C01837=1110.266,-32.356,-50.134,179.770,5.862,149.113
C01838=1110.271,-32.570,-50.123,179.770,5.858,149.112
C01839=1110.275,-32.820,-50.110,179.770,5.854,149.111
C01840=1110.280,-33.069,-50.097,179.769,5.849,149.110
C01841=1110.285,-33.319,-50.084,179.769,5.845,149.110
C01842=1110.291,-33.570,-50.072,179.769,5.841,149.109
C01843=1110.296,-33.819,-50.059,179.768,5.836,149.108
C01844=1110.301,-34.068,-50.046,179.768,5.832,149.107
C01845=1110.306,-34.318,-50.034,179.768,5.827,149.106
C01846=1110.312,-34.567,-50.021,179.767,5.822,149.105
C01847=1110.316,-34.817,-50.008,179.767,5.818,149.104
C01848=1110.321,-35.067,-49.996,179.766,5.813,149.104
C01849=1110.327,-35.317,-49.983,179.766,5.809,149.103
C01850=1110.332,-35.566,-49.971,179.766,5.805,149.102
C01851=1110.337,-35.816,-49.958,179.765,5.800,149.101
C01852=1110.342,-36.065,-49.945,179.765,5.795,149.100
C01853=1110.348,-36.315,-49.933,179.764,5.790,149.099
C01854=1110.353,-36.564,-49.921,179.763,5.786,149.098
C01855=1110.358,-36.814,-49.908,179.763,5.781,149.097
C01856=1110.362,-37.064,-49.895,179.762,5.777,149.097
C01857=1110.368,-37.314,-49.883,179.762,5.772,149.096
C01858=1110.374,-37.563,-49.870,179.762,5.767,149.095
C01859=1110.379,-37.813,-49.857,179.761,5.762,149.094
C01860=1110.384,-38.062,-49.845,179.760,5.758,149.093
C01861=1110.389,-38.312,-49.833,179.760,5.753,149.092
C01862=1110.394,-38.562,-49.820,179.759,5.749,149.091
C01863=1110.399,-38.811,-49.807,179.759,5.744,149.090
C01864=1110.404,-39.061,-49.795,179.758,5.739,149.089
C01865=1110.409,-39.311,-49.783,179.758,5.734,149.089
C01866=1110.415,-39.560,-49.770,179.758,5.730,149.088
C01867=1110.420,-39.810,-49.758,179.757,5.725,149.087
C01868=1110.425,-40.059,-49.746,179.756,5.719,149.086
C01869=1110.430,-40.309,-49.733,179.756,5.715,149.085
C01870=1110.435,-40.559,-49.721,179.755,5.710,149.084
C01871=1110.440,-40.808,-49.708,179.754,5.705,149.083
C01872=1110.446,-41.058,-49.696,179.753,5.700,149.082
C01873=1110.451,-41.308,-49.684,179.753,5.695,149.082
C01874=1110.456,-41.557,-49.671,179.752,5.690,149.081
C01875=1110.461,-41.807,-49.659,179.752,5.684,149.079
C01876=1110.466,-42.056,-49.647,179.751,5.680,149.079
C01877=1110.472,-42.306,-49.635,179.751,5.675,149.078
C01878=1110.476,-42.556,-49.622,179.750,5.669,149.077
C01879=1110.482,-42.806,-49.610,179.749,5.665,149.076
C01880=1110.486,-43.055,-49.598,179.749,5.660,149.075
C01881=1110.492,-43.305,-49.586,179.749,5.655,149.074
C01882=1110.497,-43.554,-49.573,179.750,5.651,149.073
C01883=1110.502,-43.804,-49.561,179.750,5.645,149.071
C01884=1110.507,-44.054,-49.549,179.750,5.640,149.070
C01885=1110.513,-44.304,-49.537,179.750,5.636,149.069
C01886=1110.518,-44.553,-49.524,179.750,5.631,149.068
C01887=1110.522,-44.768,-49.514,179.750,5.627,149.067
C01888=1110.526,-44.982,-49.504,179.750,5.623,149.066
C01889=1110.531,-45.197,-49.493,179.751,5.619,149.066
C01890=1110.535,-45.411,-49.482,179.751,5.615,149.065
C01891=1110.540,-45.626,-49.472,179.751,5.612,149.064
C01892=1110.545,-45.840,-49.463,179.751,5.608,149.063
C01893=1110.549,-46.055,-49.452,179.751,5.603,149.062
C01894=1110.554,-46.270,-49.441,179.751,5.598,149.061
C01895=1110.559,-46.519,-49.429,179.751,5.595,149.060
C01896=1110.564,-46.769,-49.418,179.752,5.589,149.059
C01897=1110.569,-47.019,-49.406,179.752,5.584,149.058
C01898=1110.574,-47.268,-49.393,179.752,5.580,149.057
C01899=1110.580,-47.518,-49.381,179.752,5.575,149.055
C01900=1110.585,-47.767,-49.369,179.753,5.571,149.054
C01901=1110.589,-48.017,-49.357,179.753,5.566,149.053
C01902=1110.595,-48.267,-49.345,179.752,5.561,149.052
C01903=1110.600,-48.516,-49.333,179.753,5.557,149.051
C01904=1110.605,-48.766,-49.321,179.753,5.552,149.050
C01905=1110.611,-49.016,-49.309,179.753,5.548,149.049
C01906=1110.615,-49.265,-49.297,179.753,5.542,149.048
C01907=1110.621,-49.515,-49.285,179.753,5.537,149.047
C01908=1110.626,-49.765,-49.273,179.753,5.533,149.046
C01909=1110.631,-50.014,-49.261,179.753,5.528,149.045
C01910=1110.636,-50.264,-49.249,179.754,5.523,149.043
C01911=1110.641,-50.514,-49.237,179.754,5.519,149.042
C01912=1110.647,-50.764,-49.226,179.754,5.514,149.041
C01913=1110.652,-51.013,-49.213,179.754,5.509,149.040
C01914=1110.656,-51.263,-49.202,179.755,5.505,149.039
C01915=1110.662,-51.513,-49.190,179.754,5.500,149.038
C01916=1110.667,-51.763,-49.178,179.755,5.496,149.037
C01917=1110.672,-52.012,-49.165,179.755,5.490,149.036
C01918=1110.677,-52.261,-49.154,179.755,5.486,149.035
C01919=1110.683,-52.511,-49.142,179.755,5.481,149.034
C01920=1110.688,-52.761,-49.130,179.755,5.476,149.033
C01921=1110.692,-53.010,-49.118,179.755,5.471,149.032
C01922=1110.698,-53.260,-49.106,179.756,5.467,149.031
C01923=1110.704,-53.510,-49.095,179.756,5.462,149.029
C01924=1110.709,-53.759,-49.083,179.756,5.458,149.029
C01925=1110.714,-54.009,-49.072,179.756,5.453,149.027
C01926=1110.719,-54.258,-49.059,179.756,5.448,149.026
C01927=1110.725,-54.508,-49.047,179.756,5.444,149.025
C01928=1110.729,-54.758,-49.036,179.756,5.439,149.024
C01929=1110.735,-55.008,-49.024,179.756,5.434,149.023
C01930=1110.740,-55.258,-49.012,179.757,5.430,149.022
C01931=1110.745,-55.507,-49.001,179.757,5.425,149.021
C01932=1110.750,-55.757,-48.989,179.757,5.421,149.020
C01933=1110.755,-56.006,-48.977,179.757,5.415,149.019
C01934=1110.761,-56.256,-48.965,179.757,5.410,149.018
C01935=1110.766,-56.506,-48.954,179.757,5.406,149.017
C01936=1110.771,-56.755,-48.942,179.757,5.401,149.016
C01937=1110.776,-57.005,-48.930,179.757,5.396,149.014
C01938=1110.781,-57.255,-48.919,179.758,5.392,149.014
C01939=1110.786,-57.505,-48.907,179.758,5.387,149.012
C01940=1110.792,-57.755,-48.895,179.757,5.382,149.011
C01941=1110.796,-58.004,-48.884,179.758,5.378,149.010
C01942=1110.802,-58.253,-48.872,179.758,5.373,149.009
C01943=1110.807,-58.468,-48.862,179.758,5.369,149.008
C01944=1110.811,-58.683,-48.852,179.758,5.365,149.007
C01945=1110.815,-58.898,-48.842,179.758,5.361,149.007
C01946=1110.820,-59.112,-48.832,179.758,5.357,149.006
C01947=1110.824,-59.326,-48.822,179.759,5.353,149.005
C01948=1110.829,-59.541,-48.812,179.758,5.349,149.004
C01949=1110.833,-59.756,-48.802,179.758,5.345,149.003
C01950=1110.837,-59.971,-48.792,179.759,5.341,149.002
C01951=1110.843,-60.220,-48.781,179.758,5.336,149.001
C01952=1110.848,-60.470,-48.769,179.758,5.331,149.000
C01953=1110.853,-60.720,-48.758,179.758,5.326,148.999
C01954=1110.858,-60.969,-48.746,179.757,5.321,148.998
C01955=1110.863,-61.219,-48.735,179.757,5.316,148.997
C01956=1110.869,-61.470,-48.724,179.757,5.311,148.996
C01957=1110.874,-61.719,-48.713,179.756,5.306,148.995
C01958=1110.879,-61.969,-48.701,179.755,5.300,148.994
C01959=1110.884,-62.218,-48.690,179.755,5.296,148.993
C01960=1110.890,-62.468,-48.678,179.755,5.291,148.992
C01961=1110.895,-62.717,-48.667,179.755,5.286,148.991
C01962=1110.900,-62.967,-48.655,179.754,5.281,148.990
C01963=1110.905,-63.217,-48.644,179.754,5.275,148.989
C01964=1110.910,-63.466,-48.632,179.753,5.270,148.988
C01965=1110.915,-63.716,-48.620,179.753,5.265,148.987
C01966=1110.921,-63.966,-48.610,179.753,5.260,148.986
C01967=1110.926,-64.216,-48.598,179.753,5.256,148.985
C01968=1110.931,-64.465,-48.587,179.752,5.250,148.984
C01969=1110.936,-64.715,-48.575,179.752,5.245,148.983
C01970=1110.942,-64.964,-48.564,179.752,5.240,148.982
C01971=1110.947,-65.214,-48.554,179.752,5.235,148.981
C01972=1110.952,-65.464,-48.542,179.752,5.230,148.980
C01973=1110.957,-65.713,-48.531,179.751,5.224,148.979
C01974=1110.963,-65.963,-48.519,179.751,5.219,148.978
C01975=1110.967,-66.213,-48.508,179.750,5.214,148.977
C01976=1110.972,-66.463,-48.497,179.751,5.209,148.976
C01977=1110.978,-66.712,-48.486,179.751,5.204,148.974
C01978=1110.983,-66.962,-48.474,179.750,5.199,148.973
C01979=1110.988,-67.212,-48.464,179.750,5.194,148.972
C01980=1110.994,-67.461,-48.452,179.750,5.189,148.971
C01981=1110.999,-67.711,-48.441,179.750,5.184,148.970
C01982=1111.004,-67.961,-48.430,179.750,5.178,148.969
C01983=1111.010,-68.210,-48.419,179.749,5.174,148.968
C01984=1111.015,-68.460,-48.407,179.749,5.168,148.967
C01985=1111.019,-68.710,-48.396,179.749,5.163,148.966
C01986=1111.026,-68.960,-48.385,179.749,5.158,148.965
C01987=1111.030,-69.209,-48.374,179.749,5.153,148.964
C01988=1111.035,-69.459,-48.364,179.749,5.148,148.963
C01989=1111.041,-69.709,-48.352,179.749,5.143,148.962
C01990=1111.046,-69.958,-48.341,179.749,5.138,148.960
C01991=1111.051,-70.209,-48.330,179.748,5.132,148.959
C01992=1111.056,-70.457,-48.319,179.748,5.127,148.958
C01993=1111.062,-70.707,-48.307,179.748,5.122,148.957
C01994=1111.067,-70.958,-48.297,179.748,5.117,148.956
C01995=1111.072,-71.207,-48.286,179.748,5.112,148.955
C01996=1111.077,-71.457,-48.275,179.748,5.106,148.954
C01997=1111.083,-71.706,-48.264,179.749,5.101,148.953
C01998=1111.088,-71.956,-48.253,179.748,5.097,148.952
C01999=1111.092,-72.171,-48.243,179.748,5.091,148.950
C02000=1111.097,-72.385,-48.234,179.748,5.087,148.950
C02001=1111.101,-72.601,-48.225,179.748,5.083,148.949
C02002=1111.106,-72.815,-48.215,179.748,5.078,148.948
C02003=1111.110,-73.030,-48.206,179.748,5.074,148.947
C02004=1111.114,-73.245,-48.196,179.748,5.069,148.946
C02005=1111.120,-73.459,-48.188,179.748,5.065,148.945
C02006=1111.124,-73.674,-48.178,179.748,5.060,148.944
C02007=1111.130,-73.924,-48.167,179.748,5.055,148.943
C02008=1111.134,-74.174,-48.156,179.748,5.050,148.941
C02009=1111.140,-74.423,-48.146,179.748,5.045,148.940
C02010=1111.145,-74.673,-48.135,179.748,5.040,148.939
C02011=1111.150,-74.923,-48.124,179.748,5.035,148.938
C02012=1111.156,-75.172,-48.112,179.748,5.030,148.937
C02013=1111.161,-75.422,-48.102,179.749,5.024,148.936
C02014=1111.166,-75.671,-48.091,179.749,5.019,148.935
C02015=1111.171,-75.922,-48.080,179.749,5.014,148.933
C02016=1111.176,-76.171,-48.070,179.749,5.009,148.932
C02017=1111.181,-76.421,-48.059,179.749,5.004,148.931
C02018=1111.187,-76.670,-48.049,179.749,4.999,148.930
C02019=1111.192,-76.921,-48.038,179.749,4.994,148.929
C02020=1111.198,-77.170,-48.027,179.750,4.988,148.928
C02021=1111.203,-77.420,-48.016,179.750,4.983,148.926
C02022=1111.208,-77.669,-48.005,179.750,4.978,148.925
C02023=1111.213,-77.919,-47.995,179.750,4.973,148.924
C02024=1111.219,-78.169,-47.984,179.750,4.968,148.923
C02025=1111.224,-78.419,-47.974,179.750,4.963,148.922
C02026=1111.229,-78.668,-47.963,179.751,4.958,148.920
C02027=1111.234,-78.918,-47.952,179.751,4.952,148.919
C02028=1111.240,-79.168,-47.942,179.751,4.947,148.918
C02029=1111.244,-79.417,-47.931,179.751,4.942,148.917
C02030=1111.250,-79.667,-47.921,179.751,4.937,148.916
C02031=1111.256,-79.917,-47.909,179.751,4.932,148.915
C02032=1111.261,-80.167,-47.899,179.752,4.927,148.913
C02033=1111.266,-80.417,-47.888,179.752,4.922,148.912
C02034=1111.271,-80.666,-47.878,179.752,4.916,148.911
C02035=1111.276,-80.916,-47.867,179.752,4.911,148.910
C02036=1111.282,-81.166,-47.857,179.752,4.906,148.909
C02037=1111.287,-81.415,-47.846,179.753,4.901,148.907
C02038=1111.292,-81.665,-47.835,179.753,4.895,148.906
C02039=1111.298,-81.915,-47.825,179.753,4.890,148.905
C02040=1111.303,-82.165,-47.815,179.753,4.885,148.904
C02041=1111.308,-82.414,-47.804,179.754,4.880,148.903
C02042=1111.313,-82.664,-47.794,179.754,4.876,148.901
C02043=1111.318,-82.913,-47.783,179.754,4.871,148.900
C02044=1111.323,-83.164,-47.773,179.755,4.865,148.899
C02045=1111.329,-83.413,-47.763,179.755,4.860,148.898
C02046=1111.334,-83.663,-47.752,179.755,4.855,148.897
C02047=1111.339,-83.913,-47.742,179.756,4.850,148.895
C02048=1111.345,-84.162,-47.731,179.756,4.844,148.894
C02049=1111.350,-84.412,-47.720,179.756,4.839,148.893
C02050=1111.355,-84.662,-47.710,179.757,4.835,148.892
C02051=1111.361,-84.911,-47.700,179.757,4.830,148.891
C02052=1111.366,-85.161,-47.689,179.757,4.825,148.889
C02053=1111.371,-85.411,-47.679,179.757,4.819,148.888
C02054=1111.376,-85.661,-47.669,179.757,4.814,148.887
C02055=1111.381,-85.876,-47.660,179.758,4.810,148.886
C02056=1111.385,-86.090,-47.650,179.758,4.806,148.885
C02057=1111.390,-86.305,-47.642,179.759,4.801,148.884
C02058=1111.395,-86.520,-47.633,179.759,4.797,148.883
C02059=1111.399,-86.735,-47.624,179.759,4.793,148.882
C02060=1111.403,-86.949,-47.616,179.760,4.789,148.881
C02061=1111.408,-87.165,-47.607,179.760,4.784,148.880
C02062=1111.412,-87.379,-47.598,179.760,4.780,148.879
C02063=1111.417,-87.629,-47.587,179.761,4.774,148.877
C02064=1111.423,-87.878,-47.577,179.761,4.770,148.876
C02065=1111.428,-88.128,-47.567,179.762,4.765,148.875
C02066=1111.433,-88.378,-47.556,179.762,4.760,148.874
C02067=1111.438,-88.627,-47.547,179.763,4.755,148.873
C02068=1111.444,-88.877,-47.536,179.763,4.750,148.871
C02069=1111.449,-89.127,-47.526,179.763,4.745,148.870
C02070=1111.454,-89.377,-47.516,179.764,4.740,148.869
C02071=1111.460,-89.626,-47.505,179.764,4.735,148.868
C02072=1111.465,-89.877,-47.495,179.765,4.730,148.866
C02073=1111.470,-90.126,-47.485,179.765,4.725,148.865
C02074=1111.476,-90.376,-47.476,179.766,4.721,148.864
C02075=1111.481,-90.626,-47.465,179.766,4.715,148.863
C02076=1111.486,-90.876,-47.455,179.766,4.710,148.861
C02077=1111.492,-91.125,-47.445,179.767,4.706,148.860
C02078=1111.496,-91.375,-47.435,179.767,4.700,148.859
C02079=1111.502,-91.625,-47.424,179.768,4.695,148.858
C02080=1111.507,-91.874,-47.414,179.768,4.691,148.857
C02081=1111.512,-92.125,-47.404,179.769,4.686,148.856
C02082=1111.517,-92.374,-47.394,179.769,4.681,148.854
C02083=1111.523,-92.623,-47.384,179.770,4.676,148.853
C02084=1111.529,-92.873,-47.374,179.770,4.671,148.852
C02085=1111.534,-93.124,-47.364,179.771,4.666,148.851
C02086=1111.539,-93.373,-47.354,179.771,4.661,148.849
C02087=1111.544,-93.623,-47.344,179.772,4.657,148.848
C02088=1111.549,-93.873,-47.333,179.772,4.652,148.847
C02089=1111.555,-94.122,-47.323,179.773,4.647,148.846
C02090=1111.560,-94.372,-47.314,179.773,4.642,148.845
C02091=1111.565,-94.621,-47.303,179.773,4.637,148.843
C02092=1111.571,-94.872,-47.293,179.774,4.633,148.842
C02093=1111.576,-95.121,-47.284,179.774,4.628,148.841
C02094=1111.581,-95.371,-47.274,179.775,4.622,148.840
C02095=1111.587,-95.620,-47.263,179.775,4.617,148.839
C02096=1111.592,-95.871,-47.253,179.776,4.613,148.837
C02097=1111.597,-96.120,-47.244,179.776,4.608,148.836
C02098=1111.602,-96.370,-47.234,179.776,4.603,148.835
C02099=1111.608,-96.619,-47.224,179.777,4.598,148.834
C02100=1111.613,-96.869,-47.214,179.777,4.593,148.833
C02101=1111.618,-97.120,-47.204,179.777,4.588,148.832
C02102=1111.624,-97.369,-47.194,179.777,4.583,148.830
C02103=1111.629,-97.618,-47.184,179.778,4.578,148.829
C02104=1111.634,-97.868,-47.174,179.779,4.573,148.828
C02105=1111.640,-98.119,-47.164,179.779,4.568,148.827
C02106=1111.644,-98.368,-47.155,179.779,4.563,148.826
C02107=1111.650,-98.618,-47.144,179.780,4.559,148.824
C02108=1111.655,-98.867,-47.135,179.780,4.553,148.823
C02109=1111.661,-99.117,-47.125,179.780,4.548,148.822
C02110=1111.666,-99.367,-47.115,179.780,4.543,148.821
C02111=1111.670,-99.582,-47.106,179.781,4.539,148.820
C02112=1111.675,-99.796,-47.098,179.781,4.535,148.819
C02113=1111.679,-100.012,-47.090,179.781,4.531,148.818
C02114=1111.684,-100.227,-47.081,179.782,4.527,148.817
C02115=1111.689,-100.441,-47.073,179.782,4.522,148.816
C02116=1111.693,-100.656,-47.064,179.782,4.518,148.815
C02117=1111.698,-100.871,-47.056,179.783,4.514,148.814
C02118=1111.703,-101.086,-47.048,179.783,4.510,148.813
C02119=1111.708,-101.335,-47.038,179.783,4.505,148.811
C02120=1111.714,-101.586,-47.028,179.784,4.500,148.810
C02121=1111.718,-101.836,-47.018,179.784,4.494,148.809
C02122=1111.723,-102.085,-47.008,179.785,4.490,148.808
C02123=1111.729,-102.335,-46.999,179.785,4.485,148.807
C02124=1111.734,-102.584,-46.989,179.785,4.480,148.805
C02125=1111.739,-102.834,-46.980,179.785,4.475,148.804
C02126=1111.745,-103.084,-46.970,179.786,4.469,148.803
C02127=1111.751,-103.333,-46.960,179.786,4.465,148.802
C02128=1111.755,-103.584,-46.951,179.787,4.460,148.801
C02129=1111.761,-103.834,-46.940,179.787,4.455,148.799
C02130=1111.766,-104.083,-46.931,179.787,4.450,148.798
C02131=1111.771,-104.333,-46.921,179.787,4.444,148.797
C02132=1111.777,-104.583,-46.912,179.788,4.440,148.796
C02133=1111.782,-104.832,-46.902,179.788,4.435,148.795
C02134=1111.787,-105.082,-46.893,179.789,4.430,148.794
C02135=1111.792,-105.331,-46.884,179.789,4.425,148.792
C02136=1111.798,-105.582,-46.874,179.789,4.420,148.791
C02137=1111.802,-105.831,-46.864,179.790,4.415,148.790
C02138=1111.808,-106.082,-46.855,179.790,4.410,148.789
C02139=1111.813,-106.331,-46.845,179.790,4.405,148.788
C02140=1111.819,-106.581,-46.836,179.791,4.400,148.786
C02141=1111.824,-106.830,-46.826,179.791,4.395,148.785
C02142=1111.830,-107.080,-46.816,179.791,4.389,148.784
C02143=1111.835,-107.330,-46.807,179.792,4.385,148.783
C02144=1111.841,-107.580,-46.797,179.792,4.380,148.782
C02145=1111.845,-107.829,-46.788,179.792,4.375,148.780
C02146=1111.851,-108.079,-46.779,179.793,4.370,148.779
C02147=1111.857,-108.329,-46.769,179.793,4.364,148.778
C02148=1111.861,-108.579,-46.759,179.793,4.359,148.777
C02149=1111.867,-108.829,-46.750,179.794,4.355,148.775
C02150=1111.872,-109.078,-46.740,179.795,4.349,148.774
C02151=1111.877,-109.328,-46.731,179.795,4.344,148.773
C02152=1111.883,-109.578,-46.722,179.795,4.339,148.772
C02153=1111.888,-109.828,-46.712,179.795,4.334,148.770
C02154=1111.893,-110.078,-46.703,179.796,4.329,148.769
C02155=1111.898,-110.327,-46.693,179.796,4.324,148.768
C02156=1111.903,-110.577,-46.684,179.796,4.318,148.767
C02157=1111.909,-110.827,-46.675,179.797,4.314,148.766
C02158=1111.914,-111.076,-46.665,179.797,4.309,148.764
C02159=1111.919,-111.326,-46.656,179.798,4.304,148.763
C02160=1111.925,-111.576,-46.647,179.798,4.299,148.762
C02161=1111.930,-111.826,-46.637,179.798,4.293,148.761
C02162=1111.935,-112.075,-46.628,179.799,4.288,148.759
C02163=1111.941,-112.326,-46.619,179.799,4.283,148.758
C02164=1111.946,-112.575,-46.610,179.799,4.278,148.757
C02165=1111.951,-112.825,-46.600,179.800,4.272,148.756
C02166=1111.957,-113.075,-46.591,179.800,4.267,148.755
C02167=1111.962,-113.290,-46.583,179.800,4.263,148.754
C02168=1111.966,-113.504,-46.575,179.801,4.259,148.752
C02169=1111.971,-113.719,-46.567,179.801,4.254,148.751
C02170=1111.975,-113.935,-46.559,179.802,4.250,148.750
C02171=1111.980,-114.150,-46.551,179.802,4.246,148.749
C02172=1111.985,-114.365,-46.543,179.802,4.241,148.748
C02173=1111.989,-114.579,-46.535,179.803,4.237,148.747
C02174=1111.994,-114.794,-46.527,179.802,4.232,148.746
C02175=1111.999,-115.044,-46.518,179.803,4.228,148.745
C02176=1112.004,-115.294,-46.510,179.804,4.222,148.743
C02177=1112.010,-115.544,-46.499,179.804,4.217,148.742
C02178=1112.015,-115.793,-46.490,179.804,4.212,148.741
C02179=1112.020,-116.043,-46.482,179.805,4.207,148.740
C02180=1112.026,-116.293,-46.473,179.805,4.201,148.739
C02181=1112.031,-116.543,-46.463,179.805,4.196,148.737
C02182=1112.037,-116.793,-46.454,179.806,4.191,148.736
C02183=1112.041,-117.042,-46.445,179.806,4.185,148.735
C02184=1112.047,-117.292,-46.436,179.807,4.180,148.733
C02185=1112.052,-117.542,-46.427,179.807,4.175,148.732
C02186=1112.058,-117.792,-46.417,179.807,4.170,148.731
C02187=1112.063,-118.041,-46.409,179.808,4.164,148.730
C02188=1112.069,-118.291,-46.400,179.808,4.159,148.728
C02189=1112.074,-118.541,-46.391,179.809,4.154,148.727
C02190=1112.079,-118.791,-46.382,179.809,4.149,148.726
C02191=1112.085,-119.041,-46.373,179.809,4.144,148.725
C02192=1112.090,-119.290,-46.363,179.810,4.138,148.723
C02193=1112.095,-119.540,-46.354,179.810,4.133,148.722
C02194=1112.100,-119.790,-46.345,179.810,4.128,148.721
C02195=1112.105,-120.040,-46.336,179.811,4.123,148.720
C02196=1112.111,-120.289,-46.328,179.812,4.117,148.718
C02197=1112.117,-120.539,-46.318,179.812,4.112,148.717
C02198=1112.122,-120.789,-46.309,179.812,4.107,148.716
C02199=1112.127,-121.039,-46.301,179.812,4.102,148.715
C02200=1112.132,-121.289,-46.292,179.813,4.096,148.713
C02201=1112.138,-121.539,-46.283,179.813,4.091,148.712
C02202=1112.143,-121.789,-46.274,179.814,4.086,148.711
C02203=1112.149,-122.038,-46.265,179.814,4.081,148.709
C02204=1112.154,-122.288,-46.256,179.814,4.074,148.708
C02205=1112.159,-122.537,-46.247,179.815,4.069,148.707
C02206=1112.165,-122.788,-46.238,179.815,4.064,148.706
C02207=1112.174,-123.205,-46.223,179.816,4.056,148.703
C02208=1112.182,-123.622,-46.209,179.817,4.047,148.701
C02209=1112.191,-124.039,-46.194,179.817,4.037,148.699
C02210=1112.200,-124.456,-46.179,179.818,4.028,148.697
C02211=1112.205,-124.706,-46.170,179.818,4.023,148.696
C02212=1112.211,-124.957,-46.162,179.819,4.018,148.694
C02213=1112.216,-125.206,-46.153,179.819,4.012,148.693
C02214=1112.222,-125.456,-46.145,179.820,4.007,148.692
C02215=1112.227,-125.705,-46.136,179.820,4.001,148.690
C02216=1112.232,-125.955,-46.127,179.820,3.996,148.689
C02217=1112.237,-126.205,-46.118,179.821,3.991,148.688
C02218=1112.242,-126.455,-46.109,179.821,3.985,148.686
C02219=1112.248,-126.704,-46.101,179.822,3.980,148.685
C02220=1112.254,-126.955,-46.092,179.822,3.974,148.684
C02221=1112.259,-127.204,-46.084,179.823,3.969,148.682
C02222=1112.264,-127.454,-46.075,179.823,3.963,148.681
C02223=1112.270,-127.717,-46.065,179.823,3.958,148.680
C02224=1112.276,-127.979,-46.057,179.824,3.952,148.678
C02225=1112.282,-128.242,-46.047,179.824,3.946,148.677
C02226=1112.287,-128.504,-46.038,179.825,3.940,148.676
C02227=1111.864,-128.495,-46.065,179.832,3.945,148.674
C02228=1111.859,-128.280,-46.072,179.832,3.949,148.675
C02229=1111.855,-128.065,-46.079,179.831,3.954,148.677
C02230=1111.850,-127.850,-46.086,179.831,3.958,148.677
C02231=1111.845,-127.634,-46.094,179.831,3.963,148.679
C02232=1111.841,-127.419,-46.102,179.830,3.968,148.680
C02233=1111.837,-127.205,-46.109,179.830,3.973,148.681
C02234=1111.832,-126.990,-46.117,179.830,3.978,148.682
C02235=1111.827,-126.775,-46.124,179.829,3.982,148.683
C02236=1111.822,-126.525,-46.133,179.828,3.987,148.685
C02237=1111.817,-126.275,-46.142,179.828,3.993,148.686
C02238=1111.811,-126.026,-46.150,179.828,3.999,148.687
C02239=1111.806,-125.776,-46.159,179.828,4.004,148.688
C02240=1111.800,-125.526,-46.168,179.827,4.009,148.690
C02241=1111.795,-125.276,-46.177,179.826,4.015,148.691
C02242=1111.790,-125.026,-46.186,179.826,4.020,148.692
C02243=1111.784,-124.777,-46.194,179.825,4.025,148.694
C02244=1111.779,-124.527,-46.203,179.825,4.031,148.695
C02245=1111.774,-124.277,-46.212,179.824,4.036,148.697
C02246=1111.769,-124.027,-46.220,179.824,4.041,148.698
C02247=1111.763,-123.777,-46.230,179.824,4.047,148.699
C02248=1111.757,-123.528,-46.238,179.823,4.053,148.700
C02249=1111.752,-123.278,-46.247,179.823,4.058,148.702
C02250=1111.747,-123.028,-46.256,179.823,4.063,148.703
C02251=1111.741,-122.778,-46.265,179.823,4.068,148.704
C02252=1111.736,-122.528,-46.274,179.822,4.074,148.706
C02253=1111.731,-122.278,-46.283,179.821,4.079,148.707
C02254=1111.726,-122.028,-46.292,179.821,4.084,148.708
C02255=1111.720,-121.779,-46.300,179.820,4.090,148.709
C02256=1111.715,-121.529,-46.309,179.820,4.095,148.711
C02257=1111.709,-121.279,-46.319,179.820,4.100,148.712
C02258=1111.704,-121.029,-46.327,179.820,4.105,148.713
C02259=1111.699,-120.780,-46.336,179.819,4.111,148.715
C02260=1111.694,-120.530,-46.346,179.818,4.116,148.716
C02261=1111.689,-120.280,-46.355,179.818,4.121,148.717
C02262=1111.683,-120.031,-46.364,179.817,4.127,148.718
C02263=1111.677,-119.781,-46.373,179.817,4.132,148.720
C02264=1111.672,-119.531,-46.382,179.817,4.137,148.721
C02265=1111.667,-119.281,-46.391,179.816,4.142,148.722
C02266=1111.661,-119.032,-46.400,179.816,4.147,148.723
C02267=1111.656,-118.782,-46.408,179.815,4.153,148.725
C02268=1111.650,-118.532,-46.418,179.815,4.158,148.726
C02269=1111.645,-118.282,-46.427,179.815,4.163,148.727
C02270=1111.640,-118.033,-46.436,179.815,4.168,148.728
C02271=1111.635,-117.783,-46.445,179.814,4.174,148.730
C02272=1111.630,-117.533,-46.454,179.814,4.179,148.731
C02273=1111.624,-117.283,-46.464,179.813,4.184,148.732
C02274=1111.619,-117.033,-46.473,179.813,4.189,148.733
C02275=1111.613,-116.784,-46.481,179.813,4.194,148.735
C02276=1111.608,-116.534,-46.491,179.812,4.200,148.736
C02277=1111.602,-116.284,-46.500,179.812,4.205,148.737
C02278=1111.597,-116.034,-46.509,179.811,4.210,148.739
C02279=1111.592,-115.785,-46.518,179.811,4.215,148.740
C02280=1111.587,-115.535,-46.527,179.811,4.221,148.741
C02281=1111.581,-115.285,-46.537,179.811,4.226,148.742
C02282=1111.576,-115.035,-46.546,179.810,4.231,148.743
C02283=1111.571,-114.785,-46.555,179.810,4.237,148.745
C02284=1111.566,-114.570,-46.563,179.809,4.240,148.746
C02285=1111.562,-114.356,-46.571,179.809,4.244,148.747
C02286=1111.557,-114.140,-46.579,179.809,4.250,148.748
C02287=1111.553,-113.926,-46.587,179.808,4.254,148.749
C02288=1111.548,-113.711,-46.595,179.808,4.259,148.750
C02289=1111.543,-113.495,-46.602,179.808,4.263,148.751
C02290=1111.539,-113.281,-46.611,179.807,4.267,148.752
C02291=1111.535,-113.065,-46.619,179.807,4.272,148.753
C02292=1111.529,-112.816,-46.629,179.807,4.277,148.754
C02293=1111.524,-112.566,-46.638,179.807,4.282,148.756
C02294=1111.519,-112.316,-46.647,179.806,4.287,148.757
C02295=1111.513,-112.066,-46.657,179.805,4.292,148.758
C02296=1111.508,-111.817,-46.666,179.805,4.297,148.760
C02297=1111.503,-111.567,-46.675,179.804,4.302,148.761
C02298=1111.497,-111.317,-46.685,179.804,4.308,148.762
C02299=1111.492,-111.067,-46.694,179.804,4.313,148.763
C02300=1111.486,-110.817,-46.703,179.804,4.318,148.764
C02301=1111.481,-110.568,-46.713,179.803,4.323,148.766
C02302=1111.476,-110.318,-46.722,179.803,4.327,148.767
C02303=1111.470,-110.068,-46.731,179.802,4.333,148.768
C02304=1111.465,-109.819,-46.741,179.802,4.338,148.769
C02305=1111.459,-109.568,-46.750,179.802,4.343,148.770
C02306=1111.455,-109.319,-46.760,179.802,4.348,148.772
C02307=1111.449,-109.069,-46.769,179.801,4.353,148.773
C02308=1111.443,-108.819,-46.778,179.801,4.359,148.774
C02309=1111.439,-108.570,-46.788,179.800,4.364,148.775
C02310=1111.433,-108.320,-46.798,179.800,4.368,148.777
C02311=1111.428,-108.071,-46.807,179.799,4.373,148.778
C02312=1111.423,-107.821,-46.816,179.799,4.379,148.779
C02313=1111.417,-107.571,-46.826,179.799,4.384,148.780
C02314=1111.413,-107.321,-46.836,179.799,4.389,148.781
C02315=1111.407,-107.071,-46.846,179.798,4.394,148.783
C02316=1111.402,-106.821,-46.855,179.797,4.398,148.784
C02317=1111.396,-106.572,-46.865,179.797,4.403,148.785
C02318=1111.391,-106.322,-46.874,179.797,4.409,148.786
C02319=1111.385,-106.072,-46.884,179.797,4.414,148.787
C02320=1111.380,-105.822,-46.893,179.797,4.419,148.789
C02321=1111.375,-105.573,-46.903,179.796,4.423,148.790
C02322=1111.369,-105.323,-46.912,179.795,4.428,148.791
C02323=1111.364,-105.073,-46.923,179.795,4.434,148.792
C02324=1111.359,-104.823,-46.931,179.795,4.439,148.793
C02325=1111.354,-104.573,-46.942,179.795,4.444,148.795
C02326=1111.349,-104.324,-46.951,179.794,4.448,148.796
C02327=1111.343,-104.074,-46.961,179.794,4.453,148.797
C02328=1111.338,-103.825,-46.970,179.793,4.459,148.798
C02329=1111.332,-103.575,-46.980,179.793,4.464,148.799
C02330=1111.327,-103.325,-46.990,179.793,4.469,148.801
C02331=1111.322,-103.075,-46.999,179.792,4.473,148.802
C02332=1111.317,-102.825,-47.009,179.792,4.478,148.803
C02333=1111.312,-102.576,-47.019,179.792,4.484,148.804
C02334=1111.306,-102.326,-47.028,179.792,4.489,148.805
C02335=1111.301,-102.076,-47.038,179.791,4.494,148.807
C02336=1111.295,-101.826,-47.048,179.790,4.498,148.808
C02337=1111.291,-101.576,-47.058,179.790,4.503,148.809
C02338=1111.285,-101.327,-47.068,179.790,4.509,148.810
C02339=1111.280,-101.077,-47.077,179.790,4.514,148.811
C02340=1111.275,-100.862,-47.086,179.789,4.518,148.813
C02341=1111.271,-100.647,-47.094,179.789,4.522,148.814
C02342=1111.266,-100.432,-47.103,179.788,4.526,148.815
C02343=1111.262,-100.218,-47.111,179.789,4.531,148.815
C02344=1111.257,-100.002,-47.120,179.788,4.535,148.817
C02345=1111.252,-99.787,-47.128,179.788,4.539,148.818
C02346=1111.248,-99.573,-47.136,179.787,4.543,148.819
C02347=1111.243,-99.358,-47.145,179.787,4.547,148.820
C02348=1111.238,-99.108,-47.155,179.786,4.552,148.821
C02349=1111.232,-98.858,-47.165,179.786,4.558,148.822
C02350=1111.227,-98.609,-47.174,179.786,4.563,148.823
C02351=1111.222,-98.359,-47.185,179.785,4.567,148.825
C02352=1111.217,-98.109,-47.195,179.785,4.572,148.826
C02353=1111.212,-97.859,-47.204,179.785,4.577,148.827
C02354=1111.206,-97.610,-47.214,179.785,4.582,148.828
C02355=1111.200,-97.360,-47.224,179.784,4.587,148.829
C02356=1111.196,-97.111,-47.234,179.784,4.592,148.830
C02357=1111.190,-96.860,-47.244,179.784,4.597,148.831
C02358=1111.185,-96.610,-47.254,179.783,4.602,148.833
C02359=1111.180,-96.361,-47.264,179.783,4.606,148.834
C02360=1111.174,-96.112,-47.274,179.782,4.612,148.835
C02361=1111.169,-95.861,-47.285,179.782,4.617,148.836
C02362=1111.164,-95.612,-47.293,179.781,4.621,148.837
C02363=1111.159,-95.362,-47.304,179.781,4.626,148.839
C02364=1111.153,-95.113,-47.314,179.781,4.631,148.840
C02365=1111.148,-94.862,-47.324,179.781,4.636,148.841
C02366=1111.143,-94.613,-47.334,179.780,4.641,148.842
C02367=1111.137,-94.364,-47.344,179.780,4.646,148.843
C02368=1111.132,-94.113,-47.354,179.780,4.651,148.845
C02369=1111.127,-93.863,-47.364,179.779,4.655,148.846
C02370=1111.122,-93.614,-47.374,179.779,4.661,148.847
C02371=1111.116,-93.364,-47.384,179.778,4.665,148.848
C02372=1111.111,-93.114,-47.395,179.777,4.671,148.850
C02373=1111.106,-92.865,-47.405,179.776,4.675,148.851
C02374=1111.101,-92.615,-47.415,179.776,4.680,148.852
C02375=1111.096,-92.365,-47.425,179.776,4.685,148.853
C02376=1111.090,-92.116,-47.435,179.775,4.689,148.854
C02377=1111.084,-91.866,-47.446,179.775,4.695,148.856
C02378=1111.080,-91.615,-47.455,179.774,4.699,148.857
C02379=1111.074,-91.366,-47.465,179.774,4.704,148.858
C02380=1111.069,-91.116,-47.475,179.774,4.709,148.859
C02381=1111.063,-90.867,-47.485,179.773,4.714,148.861
C02382=1111.058,-90.617,-47.496,179.772,4.719,148.862
C02383=1111.053,-90.367,-47.506,179.772,4.724,148.863
C02384=1111.048,-90.118,-47.516,179.771,4.729,148.864
C02385=1111.043,-89.868,-47.526,179.771,4.734,148.865
C02386=1111.037,-89.618,-47.537,179.771,4.739,148.866
C02387=1111.032,-89.368,-47.547,179.770,4.743,148.868
C02388=1111.026,-89.118,-47.557,179.770,4.748,148.869
C02389=1111.022,-88.869,-47.567,179.769,4.754,148.870
C02390=1111.017,-88.619,-47.578,179.769,4.759,148.871
C02391=1111.011,-88.369,-47.588,179.768,4.763,148.873
C02392=1111.005,-88.120,-47.598,179.768,4.769,148.874
C02393=1111.000,-87.869,-47.609,179.768,4.774,148.875
C02394=1110.995,-87.620,-47.619,179.768,4.779,148.876
C02395=1110.989,-87.370,-47.629,179.767,4.783,148.877
C02396=1110.986,-87.156,-47.638,179.767,4.788,148.879
C02397=1110.981,-86.941,-47.647,179.767,4.792,148.879
C02398=1110.976,-86.726,-47.656,179.766,4.797,148.881
C02399=1110.972,-86.511,-47.664,179.766,4.801,148.882
C02400=1110.967,-86.296,-47.674,179.766,4.805,148.883
C02401=1110.963,-86.082,-47.683,179.765,4.810,148.884
C02402=1110.958,-85.867,-47.692,179.765,4.814,148.885
C02403=1110.954,-85.652,-47.700,179.764,4.818,148.886
C02404=1110.948,-85.402,-47.711,179.764,4.823,148.887
C02405=1110.943,-85.152,-47.721,179.764,4.828,148.888
C02406=1110.938,-84.903,-47.731,179.764,4.834,148.889
C02407=1110.933,-84.653,-47.743,179.763,4.839,148.891
C02408=1110.927,-84.404,-47.753,179.763,4.844,148.892
C02409=1110.922,-84.154,-47.763,179.762,4.848,148.893
C02410=1110.917,-83.904,-47.774,179.762,4.854,148.894
C02411=1110.911,-83.654,-47.784,179.762,4.859,148.896
C02412=1110.906,-83.404,-47.794,179.761,4.864,148.897
C02413=1110.901,-83.155,-47.805,179.761,4.869,148.898
C02414=1110.896,-82.905,-47.816,179.761,4.874,148.899
C02415=1110.890,-82.655,-47.826,179.761,4.879,148.900
C02416=1110.885,-82.405,-47.837,179.761,4.885,148.901
C02417=1110.880,-82.155,-47.847,179.760,4.889,148.903
C02418=1110.874,-81.907,-47.858,179.760,4.894,148.904
C02419=1110.869,-81.656,-47.868,179.760,4.899,148.905
C02420=1110.864,-81.407,-47.879,179.759,4.905,148.906
C02421=1110.859,-81.156,-47.889,179.759,4.910,148.908
C02422=1110.854,-80.908,-47.900,179.759,4.915,148.909
C02423=1110.849,-80.657,-47.911,179.758,4.920,148.910
C02424=1110.843,-80.408,-47.921,179.758,4.925,148.911
C02425=1110.838,-80.158,-47.931,179.758,4.930,148.912
C02426=1110.833,-79.909,-47.942,179.758,4.936,148.913
C02427=1110.828,-79.658,-47.953,179.758,4.941,148.915
C02428=1110.822,-79.409,-47.963,179.758,4.946,148.916
C02429=1110.817,-79.159,-47.974,179.758,4.951,148.917
C02430=1110.812,-78.910,-47.985,179.757,4.956,148.918
C02431=1110.807,-78.659,-47.995,179.757,4.961,148.919
C02432=1110.802,-78.411,-48.006,179.757,4.966,148.920
C02433=1110.797,-78.160,-48.017,179.757,4.972,148.922
C02434=1110.791,-77.911,-48.027,179.757,4.977,148.923
C02435=1110.786,-77.661,-48.039,179.757,4.982,148.924
C02436=1110.780,-77.411,-48.049,179.756,4.987,148.925
C02437=1110.775,-77.161,-48.060,179.756,4.992,148.926
C02438=1110.770,-76.912,-48.071,179.756,4.997,148.927
C02439=1110.765,-76.662,-48.081,179.756,5.002,148.929
C02440=1110.759,-76.413,-48.092,179.756,5.008,148.930
C02441=1110.754,-76.163,-48.103,179.756,5.013,148.931
C02442=1110.748,-75.913,-48.113,179.756,5.018,148.932
C02443=1110.743,-75.663,-48.125,179.755,5.023,148.933
C02444=1110.738,-75.413,-48.135,179.755,5.028,148.935
C02445=1110.733,-75.164,-48.146,179.755,5.033,148.936
C02446=1110.728,-74.914,-48.157,179.755,5.039,148.937
C02447=1110.723,-74.665,-48.168,179.755,5.044,148.938
C02448=1110.717,-74.414,-48.179,179.755,5.049,148.939
C02449=1110.712,-74.165,-48.190,179.754,5.054,148.940
C02450=1110.707,-73.915,-48.200,179.755,5.059,148.941
C02451=1110.702,-73.665,-48.212,179.755,5.064,148.942
C02452=1110.697,-73.451,-48.221,179.755,5.069,148.944
C02453=1110.692,-73.236,-48.231,179.754,5.073,148.945
C02454=1110.688,-73.021,-48.239,179.755,5.078,148.946
C02455=1110.684,-72.806,-48.249,179.754,5.082,148.946
C02456=1110.679,-72.592,-48.259,179.755,5.086,148.947
C02457=1110.675,-72.377,-48.267,179.755,5.090,148.948
C02458=1110.670,-72.162,-48.277,179.754,5.095,148.949
C02459=1110.665,-71.948,-48.287,179.755,5.100,148.950
C02460=1110.660,-71.698,-48.297,179.755,5.105,148.952
C02461=1110.655,-71.449,-48.308,179.755,5.110,148.953
C02462=1110.649,-71.198,-48.320,179.755,5.115,148.954
C02463=1110.645,-70.949,-48.331,179.755,5.120,148.955
C02464=1110.639,-70.699,-48.341,179.755,5.126,148.956
C02465=1110.634,-70.449,-48.353,179.755,5.131,148.957
C02466=1110.629,-70.200,-48.364,179.755,5.135,148.958
C02467=1110.623,-69.950,-48.374,179.755,5.141,148.959
C02468=1110.619,-69.701,-48.386,179.755,5.147,148.960
C02469=1110.613,-69.451,-48.398,179.756,5.151,148.961
C02470=1110.608,-69.201,-48.408,179.755,5.156,148.963
C02471=1110.603,-68.951,-48.419,179.755,5.162,148.964
C02472=1110.598,-68.701,-48.431,179.755,5.167,148.965
C02473=1110.592,-68.452,-48.441,179.756,5.172,148.966
C02474=1110.587,-68.202,-48.452,179.755,5.177,148.967
C02475=1110.582,-67.952,-48.464,179.756,5.183,148.968
C02476=1110.576,-67.703,-48.475,179.756,5.187,148.969
C02477=1110.572,-67.453,-48.486,179.756,5.192,148.970
C02478=1110.566,-67.203,-48.498,179.757,5.197,148.971
C02479=1110.561,-66.954,-48.509,179.756,5.202,148.972
C02480=1110.556,-66.704,-48.519,179.756,5.208,148.973
C02481=1110.550,-66.454,-48.531,179.757,5.213,148.974
C02482=1110.546,-66.205,-48.542,179.757,5.218,148.976
C02483=1110.540,-65.955,-48.554,179.757,5.223,148.976
C02484=1110.535,-65.706,-48.565,179.757,5.228,148.978
C02485=1110.530,-65.455,-48.576,179.758,5.233,148.979
C02486=1110.525,-65.205,-48.588,179.758,5.238,148.980
C02487=1110.519,-64.957,-48.599,179.759,5.244,148.981
C02488=1110.514,-64.707,-48.611,179.758,5.249,148.982
C02489=1110.509,-64.457,-48.622,179.759,5.253,148.983
C02490=1110.503,-64.206,-48.633,179.759,5.259,148.984
C02491=1110.498,-63.958,-48.644,179.759,5.263,148.985
C02492=1110.493,-63.708,-48.655,179.760,5.269,148.986
C02493=1110.488,-63.458,-48.667,179.760,5.274,148.987
C02494=1110.483,-63.208,-48.678,179.760,5.279,148.988
C02495=1110.477,-62.959,-48.690,179.760,5.284,148.989
C02496=1110.473,-62.709,-48.701,179.761,5.289,148.990
C02497=1110.467,-62.460,-48.713,179.761,5.295,148.991
C02498=1110.462,-62.210,-48.724,179.762,5.299,148.992
C02499=1110.457,-61.960,-48.736,179.762,5.304,148.993
C02500=1110.451,-61.710,-48.746,179.762,5.309,148.994
C02501=1110.446,-61.460,-48.758,179.762,5.314,148.995
C02502=1110.441,-61.211,-48.770,179.763,5.320,148.996
C02503=1110.436,-60.961,-48.781,179.763,5.325,148.997
C02504=1110.431,-60.711,-48.793,179.763,5.329,148.998
C02505=1110.426,-60.461,-48.805,179.764,5.334,148.999
C02506=1110.420,-60.212,-48.816,179.764,5.339,149.000
C02507=1110.415,-59.963,-48.827,179.765,5.345,149.001
C02508=1110.411,-59.748,-48.837,179.765,5.348,149.002
C02509=1110.407,-59.533,-48.848,179.765,5.352,149.003
C02510=1110.402,-59.319,-48.858,179.765,5.356,149.004
C02511=1110.397,-59.104,-48.868,179.764,5.360,149.004
C02512=1110.393,-58.890,-48.878,179.764,5.364,149.005
C02513=1110.389,-58.675,-48.888,179.764,5.368,149.006
C02514=1110.384,-58.460,-48.898,179.764,5.373,149.007
C02515=1110.379,-58.246,-48.908,179.764,5.377,149.008
C02516=1110.375,-57.996,-48.919,179.764,5.381,149.009
C02517=1110.369,-57.746,-48.931,179.764,5.386,149.010
C02518=1110.364,-57.496,-48.943,179.764,5.391,149.011
C02519=1110.359,-57.247,-48.954,179.764,5.395,149.012
C02520=1110.354,-56.997,-48.966,179.764,5.400,149.013
C02521=1110.349,-56.747,-48.978,179.763,5.405,149.015
C02522=1110.343,-56.498,-48.989,179.763,5.409,149.016
C02523=1110.338,-56.248,-49.001,179.763,5.414,149.017
C02524=1110.333,-55.999,-49.012,179.762,5.419,149.018
C02525=1110.328,-55.749,-49.024,179.763,5.423,149.019
C02526=1110.322,-55.499,-49.036,179.763,5.429,149.020
C02527=1110.318,-55.249,-49.047,179.763,5.433,149.021
C02528=1110.313,-55.000,-49.060,179.763,5.438,149.022
C02529=1110.307,-54.750,-49.072,179.762,5.443,149.023
C02530=1110.302,-54.500,-49.083,179.762,5.447,149.024
C02531=1110.297,-54.250,-49.095,179.762,5.452,149.025
C02532=1110.292,-54.001,-49.107,179.761,5.456,149.026
C02533=1110.287,-53.752,-49.119,179.762,5.461,149.027
C02534=1110.282,-53.502,-49.131,179.762,5.466,149.028
C02535=1110.276,-53.252,-49.142,179.761,5.470,149.030
C02536=1110.271,-53.003,-49.154,179.761,5.475,149.031
C02537=1110.266,-52.753,-49.166,179.761,5.480,149.032
C02538=1110.261,-52.503,-49.178,179.761,5.485,149.033
C02539=1110.255,-52.254,-49.190,179.761,5.489,149.034
C02540=1110.250,-52.004,-49.201,179.761,5.495,149.035
C02541=1110.245,-51.754,-49.213,179.760,5.499,149.036
C02542=1110.240,-51.505,-49.226,179.761,5.504,149.037
C02543=1110.234,-51.255,-49.238,179.760,5.508,149.038
C02544=1110.230,-51.005,-49.249,179.760,5.513,149.039
C02545=1110.225,-50.756,-49.262,179.760,5.518,149.040
C02546=1110.219,-50.506,-49.274,179.760,5.522,149.041
C02547=1110.214,-50.256,-49.285,179.760,5.527,149.043
C02548=1110.209,-50.007,-49.297,179.760,5.532,149.043
C02549=1110.204,-49.757,-49.309,179.759,5.536,149.045
C02550=1110.198,-49.507,-49.321,179.759,5.541,149.046
C02551=1110.193,-49.258,-49.334,179.759,5.545,149.047
C02552=1110.188,-49.008,-49.346,179.759,5.551,149.048
C02553=1110.183,-48.758,-49.357,179.759,5.556,149.049
C02554=1110.178,-48.509,-49.370,179.758,5.560,149.050
C02555=1110.173,-48.259,-49.381,179.759,5.565,149.051
C02556=1110.167,-48.009,-49.393,179.759,5.570,149.052
C02557=1110.162,-47.760,-49.406,179.758,5.574,149.053
C02558=1110.157,-47.510,-49.417,179.758,5.579,149.054
C02559=1110.152,-47.261,-49.430,179.758,5.583,149.055
C02560=1110.147,-47.011,-49.442,179.758,5.588,149.057
C02561=1110.141,-46.761,-49.454,179.758,5.593,149.058
C02562=1110.136,-46.511,-49.466,179.758,5.597,149.059
C02563=1110.131,-46.262,-49.478,179.757,5.603,149.060
C02564=1110.127,-46.047,-49.489,179.757,5.607,149.061
C02565=1110.123,-45.832,-49.499,179.757,5.610,149.062
C02566=1110.118,-45.618,-49.510,179.757,5.614,149.063
C02567=1110.113,-45.403,-49.520,179.757,5.618,149.063
C02568=1110.109,-45.189,-49.531,179.757,5.622,149.064
C02569=1110.104,-44.975,-49.541,179.757,5.627,149.065
C02570=1110.100,-44.760,-49.551,179.757,5.631,149.066
C02571=1110.095,-44.545,-49.562,179.756,5.635,149.067
C02572=1110.090,-44.296,-49.574,179.756,5.639,149.068
C02573=1110.086,-44.046,-49.586,179.756,5.644,149.069
C02574=1110.080,-43.797,-49.598,179.756,5.649,149.071
C02575=1110.075,-43.547,-49.610,179.756,5.653,149.071
C02576=1110.070,-43.297,-49.623,179.756,5.659,149.073
C02577=1110.065,-43.047,-49.635,179.755,5.663,149.074
C02578=1110.060,-42.798,-49.648,179.755,5.668,149.075
C02579=1110.054,-42.548,-49.660,179.756,5.674,149.076
C02580=1110.049,-42.299,-49.672,179.756,5.678,149.077
C02581=1110.044,-42.049,-49.684,179.757,5.683,149.078
C02582=1110.039,-41.799,-49.697,179.758,5.689,149.079
C02583=1110.033,-41.549,-49.709,179.758,5.693,149.079
C02584=1110.028,-41.300,-49.721,179.759,5.698,149.080
C02585=1110.024,-41.050,-49.734,179.760,5.704,149.081
C02586=1110.018,-40.800,-49.746,179.760,5.708,149.082
C02587=1110.013,-40.551,-49.759,179.761,5.713,149.083
C02588=1110.008,-40.301,-49.771,179.761,5.718,149.084
C02589=1110.003,-40.051,-49.783,179.762,5.723,149.085
C02590=1109.997,-39.802,-49.796,179.763,5.728,149.086
C02591=1109.992,-39.552,-49.808,179.763,5.733,149.087
C02592=1109.987,-39.303,-49.820,179.763,5.738,149.088
C02593=1109.982,-39.053,-49.833,179.764,5.742,149.089
C02594=1109.977,-38.804,-49.846,179.764,5.747,149.089
C02595=1109.972,-38.554,-49.858,179.765,5.752,149.090
C02596=1109.967,-38.304,-49.870,179.765,5.757,149.091
C02597=1109.962,-38.055,-49.883,179.766,5.761,149.092
C02598=1109.956,-37.805,-49.895,179.767,5.766,149.093
C02599=1109.952,-37.555,-49.908,179.767,5.770,149.094
C02600=1109.947,-37.306,-49.920,179.768,5.775,149.095
C02601=1109.941,-37.056,-49.933,179.768,5.780,149.096
C02602=1109.935,-36.806,-49.945,179.768,5.785,149.096
C02603=1109.930,-36.557,-49.958,179.769,5.789,149.097
C02604=1109.926,-36.307,-49.971,179.770,5.794,149.098
C02605=1109.920,-36.057,-49.984,179.770,5.798,149.099
C02606=1109.915,-35.808,-49.996,179.771,5.803,149.100
C02607=1109.910,-35.558,-50.008,179.771,5.808,149.101
C02608=1109.905,-35.308,-50.021,179.772,5.813,149.102
C02609=1109.900,-35.059,-50.034,179.771,5.817,149.103
C02610=1109.894,-34.809,-50.047,179.772,5.821,149.104
C02611=1109.889,-34.560,-50.059,179.773,5.826,149.104
C02612=1109.884,-34.311,-50.072,179.773,5.830,149.105
C02613=1109.880,-34.061,-50.085,179.773,5.834,149.106
C02614=1109.874,-33.811,-50.097,179.774,5.839,149.107
C02615=1109.868,-33.561,-50.110,179.774,5.844,149.108
C02616=1109.864,-33.311,-50.123,179.775,5.848,149.109
C02617=1109.859,-33.062,-50.136,179.774,5.852,149.110
C02618=1109.854,-32.812,-50.148,179.775,5.857,149.110
C02619=1109.848,-32.563,-50.161,179.776,5.862,149.111
C02620=1109.844,-32.349,-50.172,179.776,5.865,149.112
C02621=1109.840,-32.134,-50.183,179.776,5.869,149.113
C02622=1109.835,-31.920,-50.194,179.776,5.873,149.114
C02623=1109.831,-31.705,-50.205,179.776,5.876,149.114
C02624=1109.827,-31.490,-50.217,179.777,5.880,149.115
C02625=1109.823,-31.276,-50.227,179.776,5.884,149.116
C02626=1109.818,-31.061,-50.239,179.777,5.888,149.117
C02627=1109.814,-30.847,-50.249,179.777,5.891,149.118
C02628=1109.808,-30.598,-50.262,179.777,5.896,149.119
C02629=1109.803,-30.348,-50.274,179.778,5.901,149.119
C02630=1109.798,-30.098,-50.288,179.777,5.905,149.120
C02631=1109.793,-29.849,-50.301,179.778,5.910,149.121
C02632=1109.787,-29.599,-50.314,179.778,5.914,149.122
C02633=1109.783,-29.349,-50.327,179.778,5.918,149.123
C02634=1109.778,-29.100,-50.339,179.778,5.922,149.124
C02635=1109.772,-28.850,-50.353,179.778,5.927,149.125
C02636=1109.767,-28.600,-50.366,179.778,5.931,149.126
C02637=1109.762,-28.351,-50.378,179.779,5.936,149.127
C02638=1109.757,-28.102,-50.391,179.778,5.940,149.128
C02639=1109.752,-27.851,-50.404,179.779,5.945,149.129
C02640=1109.747,-27.602,-50.417,179.779,5.949,149.130
C02641=1109.742,-27.353,-50.430,179.779,5.954,149.131
C02642=1109.736,-27.102,-50.443,179.778,5.958,149.132
C02643=1109.731,-26.853,-50.456,179.779,5.962,149.133
C02644=1109.726,-26.604,-50.468,179.778,5.967,149.134
C02645=1109.721,-26.354,-50.483,179.778,5.971,149.135
C02646=1109.716,-26.105,-50.495,179.778,5.976,149.136
C02647=1109.711,-25.855,-50.508,179.778,5.980,149.137
C02648=1109.706,-25.605,-50.521,179.778,5.984,149.138
C02649=1109.700,-25.356,-50.534,179.778,5.990,149.139
C02650=1109.696,-25.106,-50.547,179.779,5.994,149.140
C02651=1109.690,-24.856,-50.560,179.779,5.999,149.140
C02652=1109.686,-24.607,-50.574,179.780,6.004,149.141
C02653=1109.680,-24.357,-50.587,179.780,6.008,149.142
C02654=1109.675,-24.108,-50.600,179.781,6.013,149.143
C02655=1109.670,-23.858,-50.613,179.781,6.018,149.144
C02656=1109.665,-23.608,-50.626,179.782,6.023,149.145
C02657=1109.660,-23.359,-50.639,179.782,6.027,149.146
C02658=1109.654,-23.109,-50.653,179.783,6.032,149.147
C02659=1109.649,-22.860,-50.665,179.782,6.036,149.148
C02660=1109.644,-22.609,-50.679,179.783,6.041,149.149
C02661=1109.639,-22.361,-50.692,179.783,6.046,149.150
C02662=1109.634,-22.110,-50.706,179.784,6.051,149.151
C02663=1109.629,-21.861,-50.718,179.784,6.055,149.152
C02664=1109.624,-21.611,-50.731,179.784,6.060,149.152
C02665=1109.619,-21.362,-50.745,179.785,6.065,149.153
C02666=1109.614,-21.113,-50.758,179.785,6.069,149.154
C02667=1109.608,-20.862,-50.771,179.786,6.074,149.155
C02668=1109.604,-20.614,-50.785,179.786,6.079,149.156
C02669=1109.598,-20.363,-50.798,179.787,6.084,149.157
C02670=1109.593,-20.114,-50.811,179.787,6.088,149.158
C02671=1109.588,-19.864,-50.825,179.788,6.093,149.159
C02672=1109.583,-19.615,-50.838,179.788,6.097,149.160
C02673=1109.578,-19.365,-50.851,179.788,6.102,149.161
C02674=1109.572,-19.116,-50.865,179.789,6.106,149.161
C02675=1109.568,-18.866,-50.878,179.790,6.111,149.162
C02676=1109.563,-18.652,-50.890,179.790,6.116,149.163
C02677=1109.559,-18.437,-50.901,179.791,6.119,149.164
C02678=1109.554,-18.223,-50.912,179.790,6.123,149.165
C02679=1109.550,-18.009,-50.924,179.791,6.127,149.165
C02680=1109.546,-17.794,-50.936,179.792,6.131,149.166
C02681=1109.541,-17.579,-50.947,179.792,6.135,149.167
C02682=1109.537,-17.365,-50.959,179.793,6.139,149.167
C02683=1109.533,-17.151,-50.970,179.793,6.143,149.168
C02684=1109.528,-16.901,-50.984,179.793,6.147,149.169
C02685=1109.522,-16.652,-50.997,179.794,6.152,149.170
C02686=1109.518,-16.402,-51.011,179.794,6.157,149.171
C02687=1109.512,-16.153,-51.024,179.795,6.162,149.172
C02688=1109.507,-15.903,-51.038,179.795,6.166,149.173
C02689=1109.502,-15.653,-51.052,179.795,6.170,149.174
C02690=1109.497,-15.404,-51.065,179.796,6.175,149.174
C02691=1109.492,-15.154,-51.078,179.797,6.179,149.175
C02692=1109.487,-14.905,-51.092,179.797,6.184,149.176
C02693=1109.481,-14.655,-51.106,179.798,6.189,149.177
C02694=1109.477,-14.406,-51.119,179.798,6.194,149.178
C02695=1109.471,-14.156,-51.133,179.799,6.198,149.179
C02696=1109.467,-13.906,-51.146,179.800,6.203,149.179
C02697=1109.461,-13.657,-51.160,179.800,6.207,149.180
C02698=1109.456,-13.407,-51.174,179.800,6.211,149.181
C02699=1109.451,-13.158,-51.187,179.801,6.216,149.182
C02700=1109.446,-12.908,-51.201,179.801,6.221,149.183
C02701=1109.441,-12.658,-51.215,179.802,6.225,149.184
C02702=1109.436,-12.409,-51.229,179.803,6.230,149.185
C02703=1109.431,-12.159,-51.242,179.803,6.234,149.185
C02704=1109.426,-11.910,-51.256,179.804,6.239,149.186
C02705=1109.421,-11.660,-51.270,179.804,6.244,149.187
C02706=1109.416,-11.410,-51.283,179.805,6.247,149.188
C02707=1109.411,-11.161,-51.297,179.805,6.252,149.189
C02708=1109.406,-10.912,-51.311,179.806,6.257,149.190
C02709=1109.400,-10.661,-51.325,179.806,6.262,149.191
C02710=1109.395,-10.413,-51.338,179.807,6.266,149.191
C02711=1109.391,-10.163,-51.352,179.808,6.271,149.192
C02712=1109.385,-9.913,-51.366,179.808,6.275,149.193
C02713=1109.380,-9.664,-51.380,179.809,6.280,149.194
C02714=1109.375,-9.414,-51.394,179.809,6.284,149.195
C02715=1109.371,-9.164,-51.408,179.809,6.288,149.195
C02716=1109.365,-8.915,-51.421,179.810,6.293,149.196
C02717=1109.360,-8.665,-51.435,179.810,6.298,149.197
C02718=1109.355,-8.415,-51.450,179.811,6.302,149.198
C02719=1109.350,-8.167,-51.463,179.812,6.307,149.199
C02720=1109.345,-7.917,-51.477,179.812,6.312,149.200
C02721=1109.340,-7.667,-51.491,179.813,6.316,149.201
C02722=1109.334,-7.418,-51.505,179.813,6.320,149.201
C02723=1109.329,-7.168,-51.519,179.814,6.325,149.202
C02724=1109.324,-6.918,-51.533,179.814,6.329,149.203
C02725=1109.319,-6.670,-51.547,179.815,6.334,149.204
C02726=1109.314,-6.420,-51.561,179.816,6.338,149.205
C02727=1109.309,-6.169,-51.574,179.816,6.343,149.206
C02728=1109.304,-5.920,-51.589,179.817,6.348,149.206
C02729=1109.299,-5.671,-51.603,179.818,6.352,149.207
C02730=1109.294,-5.421,-51.617,179.818,6.357,149.208
C02731=1109.289,-5.171,-51.631,179.818,6.361,149.209
C02732=1109.284,-4.957,-51.643,179.819,6.365,149.210
C02733=1109.280,-4.743,-51.656,179.820,6.369,149.210
C02734=1109.276,-4.528,-51.667,179.820,6.372,149.211
C02735=1109.271,-4.314,-51.679,179.821,6.376,149.212
C02736=1109.267,-4.100,-51.691,179.821,6.380,149.212
C02737=1109.263,-3.886,-51.703,179.822,6.385,149.213
C02738=1109.258,-3.672,-51.715,179.822,6.388,149.214
C02739=1109.255,-3.457,-51.728,179.823,6.392,149.214
C02740=1109.249,-3.208,-51.742,179.823,6.397,149.215
C02741=1109.244,-2.958,-51.756,179.824,6.401,149.216
C02742=1109.239,-2.709,-51.770,179.825,6.406,149.217
C02743=1109.234,-2.459,-51.785,179.825,6.410,149.218
C02744=1109.229,-2.209,-51.799,179.826,6.415,149.219
C02745=1109.224,-1.960,-51.813,179.827,6.419,149.219
C02746=1109.219,-1.711,-51.827,179.827,6.423,149.220
C02747=1109.214,-1.461,-51.841,179.827,6.428,149.221
C02748=1109.209,-1.211,-51.856,179.828,6.433,149.222
C02749=1109.204,-0.961,-51.870,179.829,6.437,149.223
C02750=1109.198,-0.712,-51.884,179.829,6.442,149.224
C02751=1109.193,-0.463,-51.898,179.830,6.446,149.224
C02752=1109.188,-0.213,-51.912,179.831,6.451,149.225
C02753=1109.183,0.037,-51.927,179.831,6.455,149.226
C02754=1109.178,0.286,-51.941,179.832,6.460,149.227
C02755=1109.174,0.536,-51.956,179.832,6.465,149.228
C02756=1109.168,0.785,-51.970,179.833,6.469,149.228
C02757=1109.163,1.034,-51.984,179.834,6.474,149.229
C02758=1109.158,1.284,-51.998,179.834,6.478,149.230
C02759=1109.153,1.534,-52.013,179.834,6.483,149.231
C02760=1109.148,1.784,-52.027,179.835,6.487,149.232
C02761=1109.143,2.033,-52.042,179.836,6.492,149.233
C02762=1109.138,2.282,-52.057,179.837,6.496,149.234
C02763=1109.133,2.531,-52.071,179.838,6.501,149.234
C02764=1109.128,2.781,-52.085,179.838,6.505,149.235
C02765=1109.123,3.031,-52.099,179.839,6.510,149.236
C02766=1109.118,3.281,-52.113,179.839,6.515,149.237
C02767=1109.113,3.530,-52.128,179.840,6.519,149.238
C02768=1109.108,3.779,-52.143,179.841,6.524,149.238
C02769=1109.102,4.029,-52.158,179.841,6.529,149.239
C02770=1109.097,4.279,-52.172,179.842,6.533,149.240
C02771=1109.093,4.528,-52.187,179.843,6.538,149.241
C02772=1109.088,4.778,-52.201,179.843,6.542,149.242
C02773=1109.082,5.027,-52.215,179.843,6.546,149.243
C02774=1109.078,5.276,-52.230,179.844,6.551,149.244
C02775=1109.073,5.526,-52.244,179.845,6.555,149.244
C02776=1109.067,5.776,-52.259,179.845,6.560,149.245
C02777=1109.062,6.025,-52.274,179.846,6.565,149.246
C02778=1109.057,6.275,-52.288,179.846,6.569,149.247
C02779=1109.052,6.524,-52.303,179.847,6.574,149.248
C02780=1109.048,6.773,-52.318,179.848,6.578,149.248
C02781=1109.042,7.023,-52.333,179.849,6.583,149.249
C02782=1109.037,7.273,-52.347,179.849,6.588,149.250
C02783=1109.032,7.522,-52.362,179.850,6.593,149.251
C02784=1109.028,7.772,-52.376,179.850,6.597,149.252
C02785=1109.022,8.021,-52.392,179.851,6.602,149.253
C02786=1109.017,8.271,-52.406,179.852,6.606,149.254
C02787=1109.012,8.521,-52.420,179.852,6.611,149.254
C02788=1109.008,8.734,-52.433,179.853,6.615,149.255
C02789=1109.003,8.949,-52.446,179.853,6.619,149.256
C02790=1108.999,9.163,-52.458,179.854,6.623,149.257
C02791=1108.995,9.377,-52.472,179.854,6.627,149.258
C02792=1108.990,9.591,-52.484,179.854,6.630,149.258
C02793=1108.986,9.806,-52.496,179.855,6.635,149.259
C02794=1108.982,10.020,-52.510,179.855,6.638,149.260
C02795=1108.978,10.234,-52.522,179.855,6.642,149.260
C02796=1108.973,10.484,-52.536,179.856,6.647,149.261
C02797=1108.967,10.733,-52.552,179.856,6.651,149.262
C02798=1108.963,10.982,-52.567,179.857,6.656,149.263
C02799=1108.958,11.232,-52.581,179.857,6.660,149.264
C02800=1108.952,11.481,-52.597,179.858,6.664,149.265
C02801=1108.947,11.731,-52.611,179.859,6.669,149.265
C02802=1108.943,11.980,-52.626,179.859,6.674,149.266
C02803=1108.937,12.230,-52.641,179.860,6.678,149.267
C02804=1108.932,12.479,-52.656,179.860,6.682,149.268
C02805=1108.927,12.729,-52.670,179.861,6.687,149.269
C02806=1108.922,12.978,-52.686,179.861,6.691,149.270
C02807=1108.918,13.228,-52.701,179.862,6.696,149.271
C02808=1108.912,13.478,-52.716,179.862,6.700,149.271
C02809=1108.908,13.727,-52.731,179.863,6.704,149.272
C02810=1108.903,13.977,-52.745,179.863,6.709,149.273
C02811=1108.897,14.226,-52.761,179.864,6.714,149.274
C02812=1108.893,14.476,-52.776,179.864,6.718,149.275
C02813=1108.887,14.726,-52.791,179.865,6.722,149.275
C02814=1108.882,14.975,-52.806,179.865,6.727,149.276
C02815=1108.878,15.224,-52.821,179.866,6.731,149.277
C02816=1108.872,15.474,-52.835,179.867,6.736,149.278
C02817=1108.867,15.723,-52.850,179.867,6.740,149.279
C02818=1108.862,15.972,-52.866,179.867,6.744,149.280
C02819=1108.858,16.223,-52.881,179.868,6.749,149.280
C02820=1108.852,16.472,-52.896,179.869,6.753,149.281
C02821=1108.848,16.721,-52.911,179.870,6.758,149.282
C02822=1108.842,16.971,-52.927,179.870,6.762,149.283
C02823=1108.837,17.220,-52.941,179.871,6.766,149.284
C02824=1108.832,17.470,-52.957,179.871,6.771,149.284
C02825=1108.827,17.719,-52.972,179.872,6.775,149.285
C02826=1108.822,17.969,-52.988,179.872,6.779,149.286
C02827=1108.817,18.219,-53.002,179.873,6.784,149.287
C02828=1108.812,18.468,-53.018,179.874,6.788,149.288
C02829=1108.807,18.717,-53.033,179.874,6.793,149.288
C02830=1108.802,18.966,-53.048,179.875,6.796,149.289
C02831=1108.797,19.216,-53.063,179.875,6.801,149.290
C02832=1108.792,19.466,-53.078,179.876,6.805,149.291
C02833=1108.788,19.715,-53.093,179.877,6.810,149.292
C02834=1108.782,19.965,-53.109,179.877,6.814,149.292
C02835=1108.778,20.214,-53.124,179.878,6.818,149.293
C02836=1108.772,20.463,-53.140,179.879,6.823,149.294
C02837=1108.767,20.713,-53.155,179.879,6.827,149.295
C02838=1108.763,20.962,-53.170,179.881,6.832,149.295
C02839=1108.757,21.212,-53.185,179.880,6.836,149.296
C02840=1108.752,21.462,-53.200,179.882,6.840,149.297
C02841=1108.747,21.711,-53.216,179.882,6.845,149.298
C02842=1108.742,21.960,-53.232,179.883,6.849,149.298
C02843=1108.738,22.210,-53.247,179.883,6.853,149.299
C02844=1108.733,22.424,-53.260,179.884,6.857,149.300
C02845=1108.729,22.638,-53.273,179.885,6.861,149.301
C02846=1108.725,22.853,-53.286,179.885,6.864,149.301
C02847=1108.720,23.066,-53.300,179.886,6.867,149.302
C02848=1108.716,23.280,-53.313,179.886,6.871,149.302
C02849=1108.712,23.495,-53.326,179.887,6.875,149.303
C02850=1108.707,23.708,-53.340,179.888,6.879,149.304
C02851=1108.703,23.922,-53.353,179.888,6.882,149.304
C02852=1108.698,24.172,-53.369,179.889,6.887,149.305
C02853=1108.693,24.422,-53.384,179.890,6.891,149.306
C02854=1108.688,24.671,-53.399,179.890,6.895,149.306
C02855=1108.683,24.920,-53.415,179.891,6.900,149.307
C02856=1108.678,25.170,-53.431,179.892,6.904,149.308
C02857=1108.674,25.420,-53.446,179.893,6.908,149.309
C02858=1108.668,25.669,-53.462,179.893,6.912,149.310
C02859=1108.663,25.918,-53.477,179.894,6.916,149.310
C02860=1108.658,26.168,-53.493,179.895,6.921,149.311
C02861=1108.653,26.418,-53.508,179.896,6.925,149.312
C02862=1108.648,26.667,-53.524,179.896,6.929,149.312
C02863=1108.643,26.916,-53.539,179.897,6.933,149.313
C02864=1108.639,27.166,-53.555,179.898,6.938,149.314
C02865=1108.633,27.416,-53.570,179.899,6.942,149.315
C02866=1108.628,27.664,-53.587,179.899,6.946,149.315
C02867=1108.623,27.914,-53.603,179.900,6.950,149.316
C02868=1108.619,28.164,-53.617,179.901,6.955,149.317
C02869=1108.613,28.413,-53.633,179.902,6.959,149.317
C02870=1108.609,28.663,-53.649,179.902,6.963,149.318
C02871=1108.603,28.912,-53.665,179.903,6.967,149.319
C02872=1108.598,29.161,-53.681,179.904,6.972,149.320
C02873=1108.594,29.411,-53.696,179.905,6.976,149.320
C02874=1108.589,29.660,-53.712,179.905,6.979,149.321
C02875=1108.583,29.910,-53.727,179.907,6.984,149.322
C02876=1108.578,30.160,-53.743,179.908,6.988,149.322
C02877=1108.573,30.409,-53.760,179.908,6.993,149.323
C02878=1108.569,30.658,-53.775,179.909,6.996,149.324
C02879=1108.564,30.908,-53.791,179.910,7.001,149.324
C02880=1108.559,31.157,-53.806,179.911,7.005,149.325
C02881=1108.554,31.407,-53.823,179.912,7.009,149.326
C02882=1108.549,31.656,-53.839,179.912,7.013,149.326
C02883=1108.543,31.906,-53.854,179.913,7.017,149.327
C02884=1108.539,32.155,-53.871,179.914,7.022,149.328
C02885=1108.534,32.404,-53.886,179.915,7.026,149.329
C02886=1108.529,32.654,-53.901,179.915,7.030,149.329
C02887=1108.524,32.903,-53.918,179.916,7.034,149.330
C02888=1108.519,33.152,-53.934,179.918,7.038,149.331
C02889=1108.514,33.403,-53.950,179.919,7.042,149.331
C02890=1108.509,33.651,-53.966,179.919,7.046,149.332
C02891=1108.504,33.901,-53.982,179.920,7.050,149.333
C02892=1108.499,34.151,-53.997,179.921,7.055,149.333
C02893=1108.494,34.400,-54.014,179.922,7.059,149.334
C02894=1108.489,34.650,-54.030,179.922,7.063,149.335
C02895=1108.484,34.898,-54.046,179.923,7.067,149.335
C02896=1108.479,35.149,-54.062,179.924,7.071,149.336
C02897=1108.474,35.398,-54.078,179.925,7.076,149.337
C02898=1108.469,35.647,-54.094,179.926,7.079,149.337
C02899=1108.464,35.897,-54.110,179.927,7.084,149.338
C02900=1108.460,36.111,-54.124,179.928,7.087,149.338
C02901=1108.456,36.325,-54.137,179.929,7.091,149.339
C02902=1108.452,36.539,-54.151,179.929,7.094,149.340
C02903=1108.447,36.753,-54.164,179.930,7.098,149.340
C02904=1108.443,36.966,-54.179,179.931,7.101,149.341
C02905=1108.439,37.181,-54.192,179.932,7.104,149.341
C02906=1108.435,37.395,-54.206,179.933,7.109,149.342
C02907=1108.430,37.609,-54.220,179.934,7.112,149.342
C02908=1108.425,37.858,-54.236,179.935,7.116,149.343
C02909=1108.421,38.107,-54.253,179.935,7.120,149.344
C02910=1108.415,38.357,-54.268,179.936,7.124,149.344
C02911=1108.411,38.606,-54.285,179.937,7.128,149.345
C02912=1108.406,38.856,-54.301,179.938,7.132,149.346
C02913=1108.401,39.105,-54.317,179.939,7.136,149.346
C02914=1108.395,39.355,-54.334,179.940,7.140,149.347
C02915=1108.390,39.604,-54.350,179.941,7.145,149.348
C02916=1108.385,39.853,-54.367,179.942,7.149,149.348
C02917=1108.381,40.103,-54.382,179.942,7.152,149.349
C02918=1108.375,40.352,-54.399,179.944,7.157,149.350
C02919=1108.371,40.602,-54.415,179.945,7.161,149.350
C02920=1108.366,40.851,-54.431,179.946,7.165,149.351
C02921=1108.361,41.100,-54.448,179.946,7.169,149.352
C02922=1108.356,41.351,-54.464,179.948,7.173,149.352
C02923=1108.351,41.599,-54.480,179.949,7.177,149.353
C02924=1108.346,41.849,-54.497,179.950,7.181,149.353
C02925=1108.341,42.099,-54.513,179.950,7.185,149.354
C02926=1108.336,42.348,-54.530,179.951,7.189,149.355
C02927=1108.331,42.597,-54.546,179.952,7.193,149.355
C02928=1108.327,42.846,-54.562,179.954,7.198,149.356
C02929=1108.322,43.096,-54.578,179.954,7.201,149.356
C02930=1108.316,43.346,-54.595,179.956,7.205,149.357
C02931=1108.312,43.595,-54.612,179.957,7.209,149.358
C02932=1108.306,43.844,-54.628,179.958,7.214,149.358
C02933=1108.302,44.094,-54.644,179.959,7.218,149.359
C02934=1108.297,44.343,-54.661,179.959,7.222,149.360
C02935=1108.292,44.592,-54.677,179.961,7.226,149.360
C02936=1108.287,44.842,-54.694,179.962,7.230,149.361
C02937=1108.281,45.091,-54.710,179.963,7.234,149.361
C02938=1108.277,45.341,-54.727,179.963,7.238,149.362
C02939=1108.273,45.590,-54.743,179.965,7.242,149.362
C02940=1108.267,45.839,-54.760,179.966,7.246,149.363
C02941=1108.262,46.089,-54.777,179.967,7.250,149.364
C02942=1108.258,46.338,-54.794,179.968,7.254,149.364
C02943=1108.253,46.587,-54.810,179.969,7.258,149.365
C02944=1108.247,46.838,-54.827,179.970,7.262,149.366
C02945=1108.243,47.087,-54.843,179.971,7.266,149.366
C02946=1108.238,47.336,-54.859,179.972,7.270,149.367
C02947=1108.233,47.585,-54.876,179.973,7.274,149.367
C02948=1108.228,47.835,-54.893,179.974,7.278,149.368
C02949=1108.223,48.084,-54.910,179.975,7.282,149.369
C02950=1108.218,48.333,-54.926,179.977,7.286,149.369
C02951=1108.213,48.583,-54.944,179.977,7.290,149.370
C02952=1108.208,48.832,-54.960,179.979,7.294,149.370
C02953=1108.204,49.081,-54.977,179.980,7.298,149.371
C02954=1108.198,49.331,-54.994,179.981,7.302,149.371
C02955=1108.193,49.580,-55.010,179.982,7.306,149.372
C02956=1108.189,49.794,-55.024,179.983,7.310,149.372
C02957=1108.186,50.009,-55.039,179.984,7.313,149.373
C02958=1108.181,50.223,-55.054,179.985,7.316,149.374
C02959=1108.177,50.436,-55.068,179.986,7.319,149.374
C02960=1108.173,50.650,-55.083,179.987,7.324,149.375
C02961=1108.169,50.865,-55.096,179.988,7.327,149.375
C02962=1108.164,51.079,-55.111,179.988,7.330,149.376
C02963=1108.160,51.292,-55.126,179.989,7.333,149.376
C02964=1108.155,51.542,-55.142,179.990,7.337,149.377
C02965=1108.150,51.791,-55.159,179.992,7.342,149.377
C02966=1108.145,52.040,-55.176,179.993,7.345,149.378
C02967=1108.140,52.290,-55.193,179.994,7.349,149.378
C02968=1108.135,52.539,-55.210,179.995,7.353,149.379
C02969=1108.130,52.788,-55.226,179.996,7.357,149.379
C02970=1108.125,53.038,-55.244,179.997,7.362,149.380
C02971=1108.121,53.287,-55.261,179.998,7.366,149.381
C02972=1108.116,53.537,-55.278,179.999,7.369,149.381
C02973=1108.111,53.786,-55.294,-180.000,7.373,149.382
C02974=1108.105,54.035,-55.312,-179.998,7.377,149.382
C02975=1108.101,54.285,-55.328,-179.997,7.381,149.383
C02976=1108.096,54.534,-55.346,-179.996,7.386,149.384
C02977=1108.091,54.783,-55.363,-179.995,7.389,149.384
C02978=1108.086,55.033,-55.380,-179.994,7.393,149.385
C02979=1108.081,55.282,-55.397,-179.992,7.397,149.385
C02980=1108.076,55.532,-55.414,-179.991,7.401,149.386
C02981=1108.072,55.781,-55.431,-179.990,7.405,149.386
C02982=1108.066,56.030,-55.448,-179.989,7.409,149.387
C02983=1108.062,56.279,-55.465,-179.988,7.413,149.387
C02984=1108.056,56.529,-55.482,-179.986,7.417,149.388
C02985=1108.052,56.778,-55.499,-179.985,7.421,149.389
C02986=1108.047,57.028,-55.517,-179.984,7.425,149.389
C02987=1108.042,57.278,-55.534,-179.983,7.429,149.390
C02988=1108.037,57.526,-55.551,-179.982,7.433,149.390
C02989=1108.032,57.776,-55.568,-179.981,7.437,149.391
C02990=1108.027,58.025,-55.585,-179.979,7.441,149.391
C02991=1108.022,58.274,-55.603,-179.978,7.445,149.392
C02992=1108.017,58.524,-55.620,-179.977,7.448,149.392
C02993=1108.013,58.773,-55.637,-179.976,7.452,149.393
C02994=1108.008,59.023,-55.655,-179.974,7.456,149.393
C02995=1108.003,59.272,-55.671,-179.973,7.461,149.394
C02996=1107.997,59.521,-55.688,-179.972,7.465,149.394
C02997=1107.993,59.770,-55.706,-179.971,7.468,149.395
C02998=1107.988,60.020,-55.723,-179.970,7.472,149.396
C02999=1107.983,60.269,-55.741,-179.969,7.476,149.396
C03000=1107.978,60.519,-55.758,-179.967,7.480,149.397
C03001=1107.974,60.768,-55.776,-179.966,7.485,149.397
C03002=1107.969,61.018,-55.793,-179.964,7.488,149.398
C03003=1107.964,61.267,-55.811,-179.964,7.492,149.398
C03004=1107.959,61.516,-55.828,-179.962,7.496,149.399
C03005=1107.954,61.765,-55.846,-179.961,7.500,149.399
C03006=1107.949,62.015,-55.863,-179.960,7.504,149.400
C03007=1107.945,62.264,-55.880,-179.959,7.508,149.401
C03008=1107.939,62.513,-55.897,-179.958,7.511,149.401
C03009=1107.934,62.762,-55.915,-179.956,7.515,149.401
C03010=1107.930,63.012,-55.932,-179.955,7.520,149.402
C03011=1107.925,63.261,-55.950,-179.953,7.524,149.402
C03012=1107.921,63.476,-55.965,-179.952,7.527,149.403
C03013=1107.917,63.689,-55.979,-179.951,7.531,149.403
C03014=1107.912,63.903,-55.995,-179.950,7.534,149.404
C03015=1107.908,64.116,-56.010,-179.949,7.537,149.404
C03016=1107.903,64.330,-56.025,-179.949,7.540,149.405
C03017=1107.900,64.545,-56.039,-179.947,7.544,149.405
C03018=1107.896,64.758,-56.055,-179.946,7.547,149.406
C03019=1107.891,64.972,-56.070,-179.945,7.550,149.406
C03020=1107.887,65.221,-56.088,-179.944,7.554,149.407
C03021=1107.882,65.471,-56.105,-179.942,7.559,149.407
C03022=1107.877,65.720,-56.123,-179.941,7.563,149.408
C03023=1107.872,65.969,-56.141,-179.939,7.566,149.408
C03024=1107.866,66.219,-56.158,-179.938,7.571,149.409
C03025=1107.862,66.468,-56.175,-179.937,7.574,149.409
C03026=1107.857,66.717,-56.193,-179.936,7.578,149.410
C03027=1107.852,66.967,-56.211,-179.935,7.582,149.410
C03028=1107.847,67.216,-56.229,-179.933,7.586,149.411
C03029=1107.842,67.465,-56.247,-179.932,7.590,149.411
C03030=1107.837,67.714,-56.265,-179.930,7.594,149.412
C03031=1107.833,67.964,-56.281,-179.929,7.598,149.412
C03032=1107.829,68.214,-56.300,-179.928,7.602,149.413
C03033=1107.824,68.463,-56.318,-179.927,7.605,149.413
C03034=1107.819,68.712,-56.336,-179.926,7.610,149.414
C03035=1107.814,68.962,-56.353,-179.924,7.614,149.414
C03036=1107.809,69.211,-56.371,-179.922,7.618,149.415
C03037=1107.804,69.460,-56.389,-179.921,7.622,149.416
C03038=1107.799,69.709,-56.407,-179.920,7.626,149.416
C03039=1107.794,69.959,-56.425,-179.919,7.629,149.416
C03040=1107.789,70.208,-56.442,-179.918,7.633,149.417
C03041=1107.784,70.458,-56.460,-179.916,7.637,149.417
C03042=1107.779,70.707,-56.478,-179.915,7.641,149.418
C03043=1107.775,70.956,-56.495,-179.913,7.645,149.419
C03044=1107.770,71.205,-56.513,-179.912,7.649,149.419
C03045=1107.766,71.455,-56.532,-179.910,7.653,149.419
C03046=1107.761,71.704,-56.550,-179.909,7.657,149.420
C03047=1107.756,71.953,-56.568,-179.908,7.661,149.421
C03048=1107.751,72.202,-56.586,-179.907,7.664,149.421
C03049=1107.746,72.451,-56.604,-179.905,7.669,149.422
C03050=1107.741,72.701,-56.622,-179.904,7.673,149.422
C03051=1107.736,72.950,-56.639,-179.902,7.676,149.422
C03052=1107.731,73.200,-56.657,-179.901,7.681,149.423
C03053=1107.727,73.449,-56.675,-179.900,7.685,149.424
C03054=1107.722,73.699,-56.693,-179.898,7.688,149.424
C03055=1107.717,73.948,-56.711,-179.897,7.692,149.424
C03056=1107.711,74.197,-56.730,-179.895,7.697,149.425
C03057=1107.706,74.446,-56.748,-179.894,7.700,149.425
C03058=1107.702,74.696,-56.767,-179.893,7.704,149.426
C03059=1107.697,74.945,-56.785,-179.892,7.708,149.427
C03060=1107.692,75.194,-56.803,-179.890,7.712,149.427
C03061=1107.687,75.443,-56.821,-179.889,7.716,149.427
C03062=1107.682,75.692,-56.839,-179.887,7.720,149.428
C03063=1107.678,75.942,-56.857,-179.886,7.724,149.429
C03064=1107.673,76.191,-56.875,-179.884,7.728,149.429
C03065=1107.668,76.441,-56.893,-179.883,7.732,149.429
C03066=1107.663,76.690,-56.911,-179.882,7.736,149.430
C03067=1107.658,76.939,-56.930,-179.880,7.740,149.430
C03068=1107.655,77.153,-56.945,-179.879,7.743,149.431
C03069=1107.650,77.366,-56.961,-179.878,7.746,149.431
C03070=1107.646,77.581,-56.977,-179.878,7.749,149.432
C03071=1107.642,77.794,-56.993,-179.877,7.752,149.432
C03072=1107.637,78.008,-57.008,-179.876,7.755,149.433
C03073=1107.633,78.222,-57.024,-179.875,7.758,149.433
C03074=1107.629,78.435,-57.040,-179.874,7.761,149.434
C03075=1107.625,78.650,-57.056,-179.874,7.765,149.434
C03076=1107.620,78.899,-57.074,-179.872,7.769,149.435
C03077=1107.615,79.148,-57.092,-179.872,7.772,149.435
C03078=1107.611,79.397,-57.110,-179.870,7.776,149.436
C03079=1107.606,79.647,-57.129,-179.870,7.780,149.437
C03080=1107.601,79.896,-57.147,-179.868,7.784,149.437
C03081=1107.596,80.145,-57.165,-179.868,7.787,149.438
C03082=1107.592,80.395,-57.184,-179.866,7.791,149.438
C03083=1107.587,80.643,-57.202,-179.866,7.794,149.439
C03084=1107.581,80.893,-57.221,-179.864,7.798,149.439
C03085=1107.576,81.142,-57.239,-179.863,7.802,149.440
C03086=1107.572,81.391,-57.258,-179.862,7.806,149.440
C03087=1107.568,81.641,-57.276,-179.861,7.810,149.441
C03088=1107.562,81.890,-57.294,-179.860,7.813,149.442
C03089=1107.558,82.139,-57.313,-179.859,7.817,149.442
C03090=1107.553,82.388,-57.331,-179.858,7.821,149.443
C03091=1107.548,82.638,-57.349,-179.857,7.825,149.443
C03092=1107.543,82.887,-57.369,-179.856,7.828,149.444
C03093=1107.538,83.136,-57.387,-179.854,7.832,149.444
C03094=1107.534,83.386,-57.405,-179.854,7.836,149.445
C03095=1107.529,83.635,-57.425,-179.852,7.840,149.445
C03096=1107.524,83.884,-57.443,-179.851,7.843,149.446
C03097=1107.519,84.133,-57.461,-179.850,7.847,149.446
C03098=1107.514,84.383,-57.480,-179.849,7.851,149.447
C03099=1107.509,84.632,-57.498,-179.848,7.854,149.447
C03100=1107.505,84.881,-57.517,-179.847,7.858,149.448
C03101=1107.500,85.131,-57.536,-179.845,7.862,149.448
C03102=1107.495,85.380,-57.555,-179.844,7.866,149.449
C03103=1107.490,85.629,-57.573,-179.843,7.870,149.450
C03104=1107.485,85.878,-57.592,-179.842,7.874,149.450
C03105=1107.480,86.127,-57.610,-179.841,7.877,149.450
C03106=1107.476,86.376,-57.629,-179.840,7.881,149.451
C03107=1107.471,86.626,-57.648,-179.839,7.884,149.452
C03108=1107.466,86.875,-57.667,-179.838,7.889,149.452
C03109=1107.461,87.125,-57.685,-179.836,7.892,149.453
C03110=1107.457,87.373,-57.704,-179.835,7.896,149.453
C03111=1107.452,87.623,-57.722,-179.834,7.900,149.454
C03112=1107.447,87.872,-57.742,-179.832,7.904,149.454
C03113=1107.442,88.121,-57.760,-179.832,7.907,149.455
C03114=1107.437,88.371,-57.779,-179.830,7.911,149.455
C03115=1107.433,88.620,-57.798,-179.829,7.915,149.456
C03116=1107.428,88.870,-57.817,-179.828,7.918,149.456
C03117=1107.423,89.118,-57.836,-179.826,7.922,149.457
C03118=1107.417,89.368,-57.854,-179.825,7.926,149.457
C03119=1107.413,89.617,-57.873,-179.824,7.931,149.458
C03120=1107.408,89.866,-57.893,-179.823,7.934,149.458
C03121=1107.404,90.116,-57.911,-179.821,7.938,149.459
C03122=1107.399,90.364,-57.930,-179.820,7.941,149.459
C03123=1107.394,90.614,-57.949,-179.819,7.945,149.460
C03124=1107.390,90.827,-57.965,-179.817,7.949,149.460
C03125=1107.386,91.041,-57.981,-179.816,7.952,149.461
C03126=1107.382,91.254,-57.998,-179.816,7.955,149.461
C03127=1107.377,91.469,-58.014,-179.815,7.958,149.461
C03128=1107.374,91.683,-58.030,-179.813,7.961,149.462
C03129=1107.369,91.896,-58.046,-179.812,7.965,149.462
C03130=1107.366,92.110,-58.063,-179.811,7.968,149.463
C03131=1107.361,92.323,-58.079,-179.810,7.971,149.463
C03132=1107.356,92.572,-58.098,-179.808,7.975,149.463
C03133=1107.351,92.821,-58.118,-179.807,7.978,149.464
C03134=1107.347,93.071,-58.136,-179.806,7.982,149.465
C03135=1107.341,93.320,-58.155,-179.804,7.986,149.465
C03136=1107.337,93.569,-58.174,-179.803,7.990,149.465
C03137=1107.332,93.818,-58.194,-179.802,7.993,149.466
C03138=1107.327,94.068,-58.213,-179.801,7.997,149.466
C03139=1107.322,94.317,-58.231,-179.799,8.001,149.467
C03140=1107.318,94.567,-58.251,-179.797,8.005,149.467
C03141=1107.313,94.815,-58.270,-179.796,8.009,149.468
C03142=1107.308,95.065,-58.289,-179.795,8.012,149.468
C03143=1107.304,95.314,-58.309,-179.793,8.016,149.469
C03144=1107.299,95.563,-58.328,-179.792,8.020,149.469
C03145=1107.294,95.812,-58.347,-179.790,8.024,149.470
C03146=1107.289,96.062,-58.366,-179.789,8.027,149.470
C03147=1107.285,96.311,-58.385,-179.788,8.031,149.471
C03148=1107.279,96.560,-58.404,-179.786,8.035,149.471
C03149=1107.275,96.810,-58.424,-179.785,8.039,149.471
C03150=1107.271,97.059,-58.443,-179.783,8.043,149.472
C03151=1107.265,97.308,-58.462,-179.782,8.046,149.472
C03152=1107.260,97.557,-58.482,-179.781,8.050,149.473
C03153=1107.256,97.806,-58.501,-179.779,8.054,149.473
C03154=1107.251,98.055,-58.520,-179.777,8.058,149.474
C03155=1107.246,98.304,-58.540,-179.776,8.062,149.474
C03156=1107.242,98.553,-58.559,-179.774,8.065,149.475
C03157=1107.237,98.803,-58.578,-179.773,8.069,149.475
C03158=1107.232,99.052,-58.598,-179.772,8.072,149.475
C03159=1107.227,99.301,-58.617,-179.770,8.076,149.476
C03160=1107.223,99.551,-58.636,-179.768,8.080,149.476
C03161=1107.218,99.800,-58.656,-179.766,8.084,149.477
C03162=1107.213,100.049,-58.675,-179.765,8.088,149.477
C03163=1107.208,100.298,-58.695,-179.764,8.091,149.477
C03164=1107.203,100.548,-58.714,-179.762,8.095,149.478
C03165=1107.199,100.796,-58.734,-179.760,8.098,149.478
C03166=1107.194,101.045,-58.753,-179.759,8.102,149.479
C03167=1107.189,101.295,-58.773,-179.757,8.106,149.479
C03168=1107.184,101.544,-58.793,-179.756,8.110,149.480
C03169=1107.179,101.793,-58.812,-179.754,8.114,149.480
C03170=1107.175,102.042,-58.831,-179.753,8.117,149.480
C03171=1107.170,102.292,-58.851,-179.751,8.121,149.481
C03172=1107.165,102.540,-58.871,-179.749,8.124,149.481
C03173=1107.160,102.790,-58.890,-179.748,8.128,149.482
C03174=1107.156,103.039,-58.910,-179.746,8.132,149.482
C03175=1107.151,103.289,-58.930,-179.744,8.136,149.482
C03176=1107.146,103.538,-58.949,-179.743,8.140,149.483
C03177=1107.141,103.787,-58.969,-179.741,8.143,149.483
C03178=1107.137,104.036,-58.988,-179.739,8.147,149.483
C03179=1107.132,104.285,-59.008,-179.738,8.150,149.484
C03180=1107.127,104.499,-59.025,-179.736,8.154,149.484
C03181=1107.124,104.712,-59.042,-179.735,8.157,149.484
C03182=1107.120,104.926,-59.059,-179.733,8.159,149.485
C03183=1107.116,105.139,-59.076,-179.732,8.163,149.485
C03184=1107.111,105.353,-59.092,-179.730,8.166,149.485
C03185=1107.108,105.567,-59.109,-179.729,8.169,149.485
C03186=1107.103,105.780,-59.127,-179.727,8.173,149.486
C03187=1107.100,105.994,-59.143,-179.726,8.175,149.486
C03188=1107.094,106.243,-59.163,-179.724,8.179,149.487
C03189=1107.090,106.492,-59.183,-179.722,8.183,149.487
C03190=1107.085,106.741,-59.203,-179.721,8.187,149.487
C03191=1107.081,106.991,-59.222,-179.719,8.190,149.487
C03192=1107.075,107.239,-59.242,-179.717,8.194,149.488
C03193=1107.071,107.489,-59.262,-179.715,8.198,149.488
C03194=1107.066,107.737,-59.282,-179.714,8.201,149.489
C03195=1107.062,107.987,-59.302,-179.712,8.204,149.489
C03196=1107.057,108.237,-59.322,-179.710,8.208,149.489
C03197=1107.052,108.485,-59.342,-179.708,8.212,149.489
C03198=1107.047,108.734,-59.361,-179.707,8.215,149.490
C03199=1107.043,108.983,-59.382,-179.705,8.219,149.490
C03200=1107.037,109.233,-59.402,-179.703,8.222,149.490
C03201=1107.033,109.482,-59.422,-179.701,8.226,149.491
C03202=1107.028,109.732,-59.442,-179.699,8.230,149.491
C03203=1107.023,109.980,-59.462,-179.697,8.233,149.491
C03204=1107.018,110.230,-59.482,-179.695,8.237,149.492
C03205=1107.014,110.479,-59.502,-179.693,8.241,149.492
C03206=1107.009,110.727,-59.522,-179.691,8.244,149.492
C03207=1107.005,110.977,-59.542,-179.689,8.248,149.493
C03208=1107.000,111.226,-59.562,-179.688,8.251,149.493
C03209=1106.995,111.475,-59.582,-179.686,8.254,149.493
C03210=1106.990,111.724,-59.603,-179.684,8.258,149.493
C03211=1106.985,111.973,-59.623,-179.682,8.262,149.494
C03212=1106.980,112.223,-59.643,-179.681,8.265,149.494
C03213=1106.976,112.472,-59.663,-179.679,8.268,149.494
C03214=1106.971,112.721,-59.683,-179.677,8.272,149.495
C03215=1106.967,112.970,-59.703,-179.676,8.275,149.495
C03216=1106.962,113.219,-59.724,-179.674,8.278,149.495
C03217=1106.957,113.469,-59.744,-179.672,8.282,149.495
C03218=1106.952,113.717,-59.764,-179.671,8.285,149.496
C03219=1106.947,113.966,-59.784,-179.669,8.288,149.496
C03220=1106.943,114.215,-59.805,-179.667,8.292,149.496
C03221=1106.937,114.465,-59.825,-179.665,8.296,149.497
C03222=1106.933,114.714,-59.845,-179.664,8.299,149.497
C03223=1106.929,114.963,-59.866,-179.662,8.302,149.497
C03224=1106.924,115.212,-59.886,-179.660,8.306,149.498
C03225=1106.919,115.462,-59.906,-179.659,8.309,149.498
C03226=1106.914,115.711,-59.927,-179.657,8.312,149.498
C03227=1106.910,115.960,-59.947,-179.655,8.316,149.499
C03228=1106.905,116.209,-59.967,-179.654,8.319,149.499
C03229=1106.900,116.458,-59.988,-179.652,8.322,149.499
C03230=1106.895,116.707,-60.008,-179.650,8.326,149.499
C03231=1106.891,116.956,-60.028,-179.649,8.329,149.500
C03232=1106.886,117.206,-60.049,-179.647,8.332,149.500
C03233=1106.881,117.455,-60.070,-179.645,8.336,149.500
C03234=1106.877,117.703,-60.090,-179.643,8.340,149.501
C03235=1106.872,117.953,-60.111,-179.641,8.342,149.501
C03236=1106.868,118.166,-60.128,-179.640,8.345,149.501
C03237=1106.864,118.380,-60.145,-179.638,8.349,149.501
C03238=1106.859,118.592,-60.163,-179.637,8.352,149.502
C03239=1106.855,118.806,-60.180,-179.636,8.355,149.502
C03240=1106.851,119.020,-60.198,-179.634,8.357,149.502
C03241=1106.847,119.233,-60.216,-179.633,8.360,149.502
C03242=1106.844,119.447,-60.233,-179.631,8.363,149.503
C03243=1106.840,119.660,-60.251,-179.630,8.365,149.503
C03244=1106.834,119.909,-60.272,-179.628,8.369,149.503
C03245=1106.830,120.158,-60.292,-179.626,8.373,149.504
C03246=1106.826,120.407,-60.313,-179.624,8.376,149.504
C03247=1106.821,120.657,-60.334,-179.623,8.379,149.504
C03248=1106.817,120.906,-60.354,-179.621,8.382,149.504
C03249=1106.811,121.155,-60.375,-179.619,8.386,149.505
C03250=1106.807,121.404,-60.396,-179.617,8.389,149.505
C03251=1106.802,121.653,-60.417,-179.615,8.393,149.505
C03252=1106.797,121.902,-60.437,-179.614,8.396,149.506
C03253=1106.793,122.151,-60.457,-179.612,8.399,149.506
C03254=1106.788,122.401,-60.478,-179.610,8.403,149.506
C03255=1106.783,122.649,-60.499,-179.608,8.406,149.506
C03256=1106.778,122.899,-60.520,-179.607,8.409,149.507
C03257=1106.774,123.148,-60.540,-179.605,8.413,149.507
C03258=1106.768,123.397,-60.561,-179.603,8.416,149.507
C03259=1106.764,123.646,-60.581,-179.602,8.419,149.507
C03260=1106.760,123.895,-60.603,-179.600,8.423,149.508
C03261=1106.755,124.144,-60.624,-179.598,8.426,149.508
C03262=1106.750,124.393,-60.645,-179.597,8.429,149.508
C03263=1106.746,124.642,-60.665,-179.594,8.433,149.508
C03264=1106.741,124.892,-60.686,-179.593,8.436,149.509
C03265=1106.736,125.141,-60.706,-179.591,8.439,149.509
C03266=1106.731,125.389,-60.728,-179.589,8.443,149.509
C03267=1106.727,125.638,-60.748,-179.587,8.446,149.510
C03268=1106.722,125.888,-60.770,-179.586,8.449,149.510
C03269=1106.718,126.137,-60.790,-179.584,8.453,149.510
C03270=1106.713,126.386,-60.812,-179.582,8.456,149.511
C03271=1106.708,126.635,-60.832,-179.581,8.459,149.511
C03272=1106.703,126.884,-60.853,-179.579,8.462,149.511
C03273=1106.698,127.133,-60.874,-179.577,8.466,149.511
C03274=1106.695,127.382,-60.896,-179.575,8.470,149.512
C03275=1106.689,127.631,-60.917,-179.574,8.473,149.512
C03276=1106.684,127.881,-60.938,-179.571,8.476,149.512
C03277=1106.680,128.129,-60.959,-179.570,8.480,149.513
C03278=1106.675,128.378,-60.980,-179.568,8.483,149.513
C03279=1106.671,128.628,-61.000,-179.566,8.486,149.513
C03280=1106.666,128.877,-61.022,-179.564,8.490,149.513
C03281=1106.661,129.126,-61.043,-179.563,8.493,149.514
C03282=1106.657,129.374,-61.064,-179.561,8.496,149.514
C03283=1106.652,129.623,-61.085,-179.559,8.500,149.514
C03284=1106.647,129.873,-61.106,-179.558,8.502,149.514
C03285=1106.643,130.122,-61.127,-179.556,8.506,149.515
C03286=1106.638,130.371,-61.148,-179.554,8.510,149.515
C03287=1106.633,130.620,-61.170,-179.553,8.512,149.515
C03288=1106.628,130.869,-61.191,-179.550,8.516,149.515
C03289=1106.624,131.119,-61.212,-179.549,8.520,149.516
C03290=1106.619,131.367,-61.233,-179.547,8.523,149.516
C03291=1106.614,131.616,-61.254,-179.545,8.526,149.516
C03292=1106.610,131.830,-61.273,-179.544,8.529,149.517
C03293=1106.606,132.043,-61.291,-179.542,8.531,149.517
C03294=1106.603,132.257,-61.309,-179.540,8.535,149.517
C03295=1106.599,132.470,-61.327,-179.539,8.538,149.517
C03296=1106.594,132.683,-61.346,-179.538,8.541,149.518
C03297=1106.590,132.896,-61.364,-179.536,8.544,149.518
C03298=1106.586,133.110,-61.382,-179.535,8.546,149.518
C03299=1106.582,133.323,-61.400,-179.534,8.549,149.518
C03300=1106.578,133.573,-61.422,-179.532,8.552,149.519
C03301=1106.573,133.821,-61.443,-179.529,8.556,149.519
C03302=1106.568,134.070,-61.465,-179.528,8.560,149.519
C03303=1106.564,134.320,-61.486,-179.526,8.563,149.520
C03304=1106.559,134.568,-61.508,-179.524,8.566,149.520
C03305=1106.554,134.818,-61.528,-179.522,8.570,149.520
C03306=1106.550,135.067,-61.551,-179.521,8.573,149.520
C03307=1106.545,135.316,-61.572,-179.519,8.576,149.521
C03308=1106.540,135.565,-61.593,-179.517,8.580,149.521
C03309=1106.536,135.814,-61.615,-179.515,8.583,149.521
C03310=1106.531,136.062,-61.636,-179.514,8.586,149.522
C03311=1106.526,136.312,-61.657,-179.512,8.590,149.522
C03312=1106.522,136.561,-61.679,-179.510,8.594,149.522
C03313=1106.517,136.810,-61.701,-179.509,8.596,149.523
C03314=1106.512,137.058,-61.723,-179.507,8.600,149.523
C03315=1106.508,137.308,-61.744,-179.505,8.603,149.523
C03316=1106.503,137.557,-61.766,-179.503,8.607,149.523
C03317=1106.499,137.805,-61.787,-179.502,8.610,149.524
C03318=1106.494,138.055,-61.809,-179.500,8.613,149.524
C03319=1106.489,138.304,-61.830,-179.498,8.617,149.524
C03320=1106.485,138.553,-61.852,-179.497,8.620,149.525
C03321=1106.480,138.802,-61.874,-179.494,8.623,149.525
C03322=1106.475,139.051,-61.895,-179.493,8.627,149.525
C03323=1106.471,139.300,-61.917,-179.491,8.631,149.525
C03324=1106.466,139.549,-61.938,-179.489,8.633,149.526
C03325=1106.461,139.798,-61.960,-179.488,8.637,149.526
C03326=1106.457,140.047,-61.982,-179.486,8.641,149.526
C03327=1106.452,140.296,-62.004,-179.483,8.644,149.527
C03328=1106.447,140.545,-62.026,-179.482,8.647,149.527
C03329=1106.443,140.794,-62.047,-179.480,8.651,149.527
C03330=1106.438,141.043,-62.069,-179.479,8.655,149.528
C03331=1106.433,141.292,-62.091,-179.477,8.658,149.528
C03332=1106.429,141.541,-62.113,-179.475,8.661,149.528
C03333=1106.424,141.790,-62.135,-179.474,8.665,149.529
C03334=1106.420,142.040,-62.156,-179.472,8.668,149.529
C03335=1106.415,142.288,-62.178,-179.469,8.672,149.529
C03336=1106.410,142.537,-62.200,-179.468,8.675,149.530
C03337=1106.406,142.786,-62.222,-179.466,8.678,149.530
C03338=1106.401,143.035,-62.243,-179.465,8.682,149.530
C03339=1106.397,143.284,-62.265,-179.463,8.686,149.530
C03340=1106.392,143.533,-62.287,-179.462,8.689,149.531
C03341=1106.387,143.782,-62.309,-179.460,8.692,149.531
C03342=1106.383,144.031,-62.331,-179.458,8.696,149.531
C03343=1106.378,144.281,-62.353,-179.456,8.700,149.532
C03344=1106.373,144.529,-62.376,-179.454,8.702,149.532
C03345=1106.369,144.778,-62.398,-179.453,8.706,149.532
C03346=1106.364,145.027,-62.420,-179.451,8.710,149.533
C03347=1106.360,145.276,-62.442,-179.449,8.714,149.533
C03348=1106.355,145.489,-62.460,-179.448,8.716,149.533
C03349=1106.352,145.703,-62.479,-179.446,8.719,149.534
C03350=1106.347,145.916,-62.498,-179.444,8.723,149.534
C03351=1106.344,146.129,-62.517,-179.443,8.725,149.534
C03352=1106.339,146.343,-62.536,-179.441,8.728,149.534
C03353=1106.336,146.555,-62.555,-179.440,8.732,149.535
C03354=1106.331,146.769,-62.574,-179.438,8.735,149.535
C03355=1106.328,146.982,-62.593,-179.437,8.737,149.535
C03356=1106.323,147.231,-62.615,-179.435,8.741,149.535
C03357=1106.318,147.480,-62.637,-179.432,8.744,149.536
C03358=1106.313,147.729,-62.659,-179.431,8.748,149.536
C03359=1106.309,147.978,-62.681,-179.429,8.752,149.536
C03360=1106.305,148.227,-62.704,-179.427,8.755,149.537
C03361=1106.300,148.476,-62.726,-179.425,8.758,149.537
C03362=1106.295,148.725,-62.748,-179.423,8.761,149.537
C03363=1106.290,148.974,-62.770,-179.422,8.765,149.538
C03364=1106.286,149.223,-62.793,-179.419,8.769,149.538
C03365=1106.281,149.472,-62.815,-179.417,8.772,149.538
C03366=1106.277,149.721,-62.837,-179.415,8.776,149.538
C03367=1106.273,149.970,-62.860,-179.414,8.778,149.538
C03368=1106.268,150.218,-62.881,-179.412,8.782,149.539
C03369=1106.263,150.468,-62.904,-179.410,8.785,149.539
C03370=1106.259,150.717,-62.927,-179.408,8.789,149.539
C03371=1106.254,150.965,-62.948,-179.406,8.792,149.539
C03372=1106.249,151.215,-62.971,-179.403,8.796,149.540
C03373=1106.244,151.463,-62.993,-179.402,8.798,149.540
C03374=1106.240,151.712,-63.015,-179.400,8.802,149.540
C03375=1106.235,151.961,-63.039,-179.398,8.805,149.540
C03376=1106.230,152.210,-63.060,-179.396,8.809,149.541
C03377=1106.226,152.459,-63.083,-179.394,8.812,149.541
C03378=1106.222,152.708,-63.106,-179.392,8.815,149.541
C03379=1106.217,152.957,-63.128,-179.390,8.819,149.541
C03380=1106.212,153.206,-63.151,-179.388,8.822,149.542
C03381=1106.208,153.455,-63.173,-179.386,8.826,149.542
C03382=1106.203,153.703,-63.195,-179.385,8.828,149.542
C03383=1106.198,153.953,-63.218,-179.382,8.832,149.542
C03384=1106.194,154.202,-63.241,-179.380,8.835,149.543
C03385=1106.189,154.451,-63.263,-179.378,8.839,149.543
C03386=1106.185,154.699,-63.286,-179.377,8.841,149.543
C03387=1106.180,154.949,-63.308,-179.374,8.845,149.543
C03388=1106.176,155.198,-63.331,-179.372,8.848,149.543
C03389=1106.171,155.446,-63.353,-179.370,8.852,149.544
C03390=1106.166,155.696,-63.376,-179.369,8.854,149.544
C03391=1106.162,155.944,-63.399,-179.367,8.858,149.544
C03392=1106.156,156.193,-63.421,-179.365,8.861,149.544
C03393=1106.153,156.442,-63.444,-179.362,8.864,149.544
C03394=1106.148,156.692,-63.467,-179.361,8.867,149.545
C03395=1106.144,156.940,-63.489,-179.358,8.871,149.545
C03396=1106.138,157.189,-63.512,-179.356,8.874,149.545
C03397=1106.134,157.438,-63.535,-179.354,8.876,149.545
C03398=1106.129,157.687,-63.558,-179.352,8.880,149.545
C03399=1106.125,157.936,-63.581,-179.350,8.883,149.545
C03400=1106.120,158.185,-63.603,-179.348,8.887,149.546
C03401=1106.116,158.433,-63.626,-179.346,8.889,149.546
C03402=1106.111,158.682,-63.649,-179.344,8.893,149.546
C03403=1106.106,158.931,-63.672,-179.342,8.896,149.546
C03404=1106.103,159.144,-63.691,-179.340,8.898,149.546
C03405=1106.099,159.358,-63.711,-179.339,8.901,149.547
C03406=1106.095,159.570,-63.730,-179.337,8.903,149.547
C03407=1106.091,159.784,-63.750,-179.335,8.906,149.547
C03408=1106.087,159.998,-63.770,-179.333,8.909,149.547
C03409=1106.083,160.210,-63.790,-179.332,8.912,149.547
C03410=1106.079,160.424,-63.809,-179.330,8.914,149.547
C03411=1106.075,160.636,-63.828,-179.328,8.917,149.547
C03412=1106.071,160.885,-63.852,-179.326,8.921,149.548
C03413=1106.066,161.135,-63.875,-179.324,8.924,149.548
C03414=1106.062,161.384,-63.897,-179.322,8.926,149.548
C03415=1106.057,161.633,-63.920,-179.320,8.929,149.548
C03416=1106.052,161.881,-63.943,-179.318,8.933,149.548
C03417=1106.048,162.130,-63.966,-179.316,8.936,149.548
C03418=1106.043,162.379,-63.989,-179.314,8.939,149.548
C03419=1106.038,162.628,-64.013,-179.311,8.942,149.549
C03420=1106.034,162.877,-64.036,-179.310,8.945,149.549
C03421=1106.030,163.126,-64.059,-179.307,8.948,149.549
C03422=1106.025,163.375,-64.082,-179.305,8.951,149.549
C03423=1106.021,163.624,-64.105,-179.304,8.954,149.549
C03424=1106.016,163.872,-64.128,-179.301,8.957,149.549
C03425=1106.011,164.121,-64.151,-179.299,8.960,149.549
C03426=1106.007,164.370,-64.174,-179.297,8.963,149.549
C03427=1106.002,164.619,-64.198,-179.295,8.966,149.550
C03428=1105.997,164.868,-64.221,-179.292,8.969,149.550
C03429=1105.993,165.117,-64.244,-179.291,8.972,149.550
C03430=1105.989,165.365,-64.267,-179.288,8.975,149.550
C03431=1105.984,165.614,-64.290,-179.286,8.979,149.550
C03432=1105.979,165.863,-64.314,-179.284,8.981,149.550
C03433=1105.975,166.113,-64.337,-179.282,8.985,149.551
C03434=1105.970,166.362,-64.360,-179.280,8.988,149.551
C03435=1105.965,166.610,-64.383,-179.278,8.990,149.551
C03436=1105.961,166.859,-64.406,-179.276,8.993,149.551
C03437=1105.956,167.108,-64.430,-179.273,8.997,149.551
C03438=1105.951,167.357,-64.453,-179.272,8.999,149.551
C03439=1105.947,167.606,-64.476,-179.269,9.002,149.551
C03440=1105.943,167.854,-64.499,-179.267,9.006,149.551
C03441=1105.938,168.103,-64.523,-179.265,9.008,149.551
C03442=1105.934,168.352,-64.546,-179.263,9.011,149.551
C03443=1105.929,168.601,-64.570,-179.261,9.015,149.552
C03444=1105.924,168.850,-64.593,-179.259,9.017,149.552
C03445=1105.920,169.099,-64.617,-179.257,9.021,149.552
C03446=1105.915,169.347,-64.641,-179.255,9.023,149.552
C03447=1105.910,169.596,-64.664,-179.252,9.026,149.552
C03448=1105.906,169.845,-64.687,-179.250,9.030,149.552
C03449=1105.902,170.094,-64.710,-179.248,9.032,149.552
C03450=1105.897,170.343,-64.734,-179.246,9.035,149.553
C03451=1105.893,170.592,-64.758,-179.244,9.038,149.553
C03452=1105.888,170.841,-64.781,-179.242,9.041,149.553
C03453=1105.883,171.090,-64.804,-179.240,9.044,149.553
C03454=1105.879,171.338,-64.828,-179.237,9.047,149.553
C03455=1105.874,171.587,-64.852,-179.235,9.050,149.553
C03456=1105.869,171.836,-64.875,-179.233,9.053,149.553
C03457=1105.865,172.085,-64.899,-179.231,9.056,149.553
C03458=1105.860,172.334,-64.922,-179.229,9.059,149.553
C03459=1105.856,172.583,-64.946,-179.227,9.062,149.554
C03460=1105.852,172.796,-64.966,-179.225,9.064,149.554
C03461=1105.849,173.008,-64.987,-179.223,9.067,149.554
C03462=1105.844,173.222,-65.007,-179.222,9.070,149.554
C03463=1105.840,173.435,-65.027,-179.220,9.072,149.554
C03464=1105.836,173.648,-65.047,-179.217,9.075,149.554
C03465=1105.833,173.861,-65.068,-179.215,9.077,149.554
C03466=1105.829,174.074,-65.088,-179.214,9.080,149.554
C03467=1105.824,174.287,-65.108,-179.212,9.082,149.554
C03468=1105.820,174.536,-65.132,-179.209,9.085,149.554
C03469=1105.816,174.785,-65.156,-179.208,9.088,149.555
C03470=1105.811,175.034,-65.180,-179.205,9.091,149.555
C03471=1105.807,175.283,-65.204,-179.204,9.094,149.555
C03472=1105.802,175.531,-65.228,-179.201,9.097,149.555
C03473=1105.798,175.780,-65.251,-179.199,9.100,149.555
C03474=1105.793,176.029,-65.275,-179.197,9.103,149.555
C03475=1105.789,176.278,-65.298,-179.195,9.106,149.555
C03476=1105.784,176.526,-65.322,-179.192,9.109,149.555
C03477=1105.780,176.776,-65.346,-179.191,9.111,149.555
C03478=1105.776,177.024,-65.370,-179.188,9.115,149.555
C03479=1105.771,177.273,-65.395,-179.186,9.118,149.556
C03480=1105.766,177.522,-65.418,-179.184,9.120,149.556
C03481=1105.761,177.770,-65.442,-179.182,9.124,149.556
C03482=1105.757,178.019,-65.466,-179.179,9.127,149.556
C03483=1105.753,178.269,-65.490,-179.178,9.129,149.556
C03484=1105.749,178.517,-65.514,-179.175,9.132,149.556
C03485=1105.744,178.766,-65.538,-179.173,9.136,149.556
C03486=1105.739,179.015,-65.562,-179.171,9.138,149.556
C03487=1105.734,179.263,-65.586,-179.169,9.141,149.556
C03488=1105.730,179.512,-65.610,-179.166,9.145,149.557
C03489=1105.726,179.761,-65.634,-179.165,9.147,149.557
C03490=1105.721,180.010,-65.658,-179.162,9.150,149.557
C03491=1105.716,180.258,-65.683,-179.160,9.154,149.557
C03492=1105.712,180.507,-65.706,-179.158,9.156,149.557
C03493=1105.708,180.757,-65.731,-179.156,9.159,149.557
C03494=1105.703,181.005,-65.755,-179.153,9.162,149.557
C03495=1105.699,181.253,-65.779,-179.151,9.165,149.557
C03496=1105.694,181.503,-65.803,-179.149,9.168,149.557
C03497=1105.689,181.751,-65.827,-179.146,9.171,149.557
C03498=1105.685,182.000,-65.851,-179.145,9.174,149.557
C03499=1105.680,182.249,-65.876,-179.142,9.177,149.557
C03500=1105.676,182.497,-65.900,-179.140,9.180,149.557
C03501=1105.671,182.746,-65.923,-179.138,9.182,149.557
C03502=1105.667,182.996,-65.948,-179.135,9.185,149.558
C03503=1105.662,183.244,-65.972,-179.133,9.189,149.558
C03504=1105.658,183.493,-65.997,-179.131,9.191,149.558
C03505=1105.654,183.742,-66.021,-179.129,9.194,149.558
C03506=1105.649,183.990,-66.046,-179.127,9.196,149.558
C03507=1105.645,184.239,-66.070,-179.124,9.200,149.558
C03508=1105.640,184.487,-66.094,-179.122,9.203,149.558
C03509=1105.636,184.737,-66.119,-179.120,9.205,149.558
C03510=1105.631,184.985,-66.143,-179.117,9.208,149.558
C03511=1105.626,185.234,-66.168,-179.115,9.211,149.558
C03512=1105.622,185.483,-66.192,-179.113,9.214,149.558
C03513=1105.618,185.731,-66.216,-179.110,9.217,149.558
C03514=1105.612,185.981,-66.240,-179.108,9.219,149.558
C03515=1105.609,186.229,-66.265,-179.106,9.222,149.558
C03516=1105.601,186.618,-66.303,-179.102,9.227,149.558
C03517=1105.594,187.006,-66.341,-179.099,9.231,149.558
C03518=1105.587,187.394,-66.380,-179.095,9.235,149.558
C03519=1105.580,187.784,-66.418,-179.091,9.240,149.559
C03520=1105.576,188.032,-66.442,-179.090,9.242,149.559
C03521=1105.572,188.280,-66.467,-179.087,9.245,149.559
C03522=1105.567,188.529,-66.492,-179.084,9.249,149.559
C03523=1105.563,188.778,-66.516,-179.083,9.251,149.559
C03524=1105.558,189.026,-66.541,-179.080,9.254,149.559
C03525=1105.554,189.275,-66.565,-179.078,9.256,149.559
C03526=1105.549,189.524,-66.590,-179.076,9.259,149.559
C03527=1105.544,189.774,-66.615,-179.073,9.263,149.559
C03528=1105.540,190.021,-66.640,-179.071,9.265,149.559
C03529=1105.535,190.270,-66.664,-179.069,9.268,149.559
C03530=1105.531,190.519,-66.689,-179.066,9.271,149.559
C03531=1105.526,190.768,-66.713,-179.064,9.273,149.559
C03532=1105.522,191.017,-66.738,-179.062,9.277,149.559
C03533=1105.517,191.265,-66.763,-179.060,9.279,149.559
C03534=1105.514,191.514,-66.788,-179.057,9.282,149.559
C03535=1105.508,191.763,-66.812,-179.055,9.285,149.559
C03536=1105.504,192.011,-66.838,-179.053,9.287,149.559
C03537=1105.500,192.260,-66.862,-179.050,9.291,149.559
C03538=1105.495,192.509,-66.887,-179.048,9.294,149.559
C03539=1105.491,192.758,-66.911,-179.046,9.296,149.559
C03540=1105.486,193.006,-66.937,-179.043,9.299,149.560
C03541=1105.481,193.256,-66.962,-179.041,9.302,149.560
C03542=1105.477,193.504,-66.986,-179.039,9.305,149.560
C03543=1105.473,193.753,-67.011,-179.037,9.308,149.560
C03544=1105.468,194.002,-67.036,-179.034,9.311,149.560
C03545=1105.464,194.250,-67.061,-179.032,9.313,149.560
C03546=1105.459,194.499,-67.086,-179.030,9.316,149.560
C03547=1105.455,194.748,-67.111,-179.028,9.320,149.560
C03548=1105.220,184.488,-66.149,-179.120,9.204,149.558
C03549=1105.224,184.240,-66.125,-179.122,9.200,149.558
C03550=1105.229,183.990,-66.100,-179.124,9.198,149.558
C03551=1105.233,183.742,-66.076,-179.127,9.195,149.557
C03552=1105.237,183.493,-66.052,-179.129,9.192,149.557
C03553=1105.242,183.243,-66.028,-179.131,9.190,149.557
C03554=1105.247,182.995,-66.004,-179.133,9.186,149.557
C03555=1105.251,182.746,-65.980,-179.136,9.183,149.557
C03556=1105.256,182.498,-65.955,-179.138,9.181,149.557
C03557=1105.260,182.249,-65.931,-179.140,9.178,149.557
C03558=1105.264,182.000,-65.906,-179.142,9.175,149.557
C03559=1105.270,181.751,-65.883,-179.144,9.172,149.557
C03560=1105.274,181.502,-65.858,-179.147,9.169,149.557
C03561=1105.278,181.253,-65.834,-179.149,9.167,149.557
C03562=1105.282,181.005,-65.810,-179.151,9.163,149.557
C03563=1105.288,180.756,-65.785,-179.153,9.160,149.557
C03564=1105.292,180.507,-65.762,-179.155,9.158,149.557
C03565=1105.296,180.258,-65.737,-179.158,9.155,149.556
C03566=1105.300,180.010,-65.713,-179.160,9.151,149.556
C03567=1105.305,179.761,-65.689,-179.162,9.149,149.556
C03568=1105.310,179.512,-65.665,-179.164,9.146,149.556
C03569=1105.315,179.263,-65.641,-179.167,9.143,149.556
C03570=1105.319,179.014,-65.617,-179.169,9.140,149.556
C03571=1105.323,178.765,-65.593,-179.171,9.137,149.556
C03572=1105.328,178.517,-65.569,-179.173,9.134,149.556
C03573=1105.333,178.268,-65.545,-179.175,9.131,149.556
C03574=1105.337,178.019,-65.521,-179.177,9.128,149.555
C03575=1105.341,177.770,-65.497,-179.180,9.125,149.555
C03576=1105.346,177.522,-65.473,-179.182,9.122,149.555
C03577=1105.350,177.273,-65.450,-179.184,9.119,149.555
C03578=1105.355,177.024,-65.425,-179.186,9.116,149.555
C03579=1105.359,176.775,-65.402,-179.188,9.113,149.555
C03580=1105.364,176.527,-65.378,-179.190,9.110,149.555
C03581=1105.369,176.277,-65.354,-179.193,9.107,149.555
C03582=1105.373,176.028,-65.330,-179.195,9.104,149.555
C03583=1105.377,175.780,-65.306,-179.197,9.101,149.554
C03584=1105.382,175.531,-65.282,-179.199,9.098,149.554
C03585=1105.387,175.282,-65.258,-179.201,9.096,149.554
C03586=1105.391,175.033,-65.235,-179.203,9.092,149.554
C03587=1105.396,174.785,-65.211,-179.205,9.090,149.554
C03588=1105.400,174.536,-65.187,-179.208,9.087,149.554
C03589=1105.404,174.292,-65.164,-179.210,9.083,149.554
C03590=1105.409,174.049,-65.141,-179.212,9.081,149.554
C03591=1105.413,173.805,-65.118,-179.214,9.078,149.554
C03592=1105.418,173.562,-65.094,-179.216,9.075,149.554
C03593=1105.422,173.317,-65.071,-179.218,9.072,149.553
C03594=1105.427,173.074,-65.048,-179.221,9.069,149.553
C03595=1105.431,172.831,-65.024,-179.222,9.066,149.553
C03596=1105.436,172.587,-65.002,-179.225,9.063,149.553
C03597=1105.440,172.337,-64.978,-179.227,9.061,149.553
C03598=1105.444,172.089,-64.954,-179.229,9.057,149.553
C03599=1105.449,171.840,-64.930,-179.231,9.054,149.553
C03600=1105.454,171.591,-64.907,-179.233,9.052,149.553
C03601=1105.458,171.342,-64.883,-179.235,9.048,149.553
C03602=1105.463,171.093,-64.860,-179.238,9.045,149.553
C03603=1105.467,170.844,-64.836,-179.240,9.043,149.552
C03604=1105.472,170.596,-64.812,-179.242,9.039,149.552
C03605=1105.477,170.347,-64.789,-179.244,9.037,149.552
C03606=1105.481,170.098,-64.766,-179.246,9.034,149.552
C03607=1105.486,169.849,-64.742,-179.248,9.030,149.552
C03608=1105.490,169.600,-64.718,-179.250,9.028,149.552
C03609=1105.495,169.351,-64.695,-179.252,9.025,149.552
C03610=1105.499,169.103,-64.672,-179.255,9.021,149.552
C03611=1105.504,168.854,-64.649,-179.257,9.019,149.552
C03612=1105.508,168.605,-64.625,-179.259,9.016,149.551
C03613=1105.513,168.356,-64.601,-179.261,9.013,149.551
C03614=1105.517,168.107,-64.578,-179.263,9.010,149.551
C03615=1105.522,167.858,-64.554,-179.265,9.007,149.551
C03616=1105.527,167.609,-64.531,-179.268,9.004,149.551
C03617=1105.532,167.360,-64.508,-179.269,9.001,149.551
C03618=1105.536,167.111,-64.485,-179.272,8.998,149.551
C03619=1105.541,166.863,-64.462,-179.274,8.994,149.550
C03620=1105.545,166.615,-64.438,-179.276,8.992,149.550
C03621=1105.550,166.366,-64.415,-179.278,8.988,149.550
C03622=1105.555,166.116,-64.391,-179.280,8.985,149.550
C03623=1105.559,165.868,-64.368,-179.282,8.983,149.550
C03624=1105.563,165.619,-64.345,-179.284,8.980,149.550
C03625=1105.568,165.370,-64.322,-179.286,8.977,149.550
C03626=1105.573,165.121,-64.298,-179.288,8.974,149.550
C03627=1105.577,164.872,-64.275,-179.291,8.971,149.550
C03628=1105.581,164.623,-64.252,-179.292,8.968,149.549
C03629=1105.586,164.374,-64.229,-179.295,8.965,149.549
C03630=1105.591,164.125,-64.206,-179.297,8.961,149.549
C03631=1105.595,163.877,-64.183,-179.299,8.959,149.549
C03632=1105.600,163.628,-64.160,-179.301,8.955,149.549
C03633=1105.605,163.379,-64.136,-179.303,8.952,149.549
C03634=1105.609,163.130,-64.113,-179.305,8.950,149.548
C03635=1105.613,162.881,-64.090,-179.307,8.946,149.548
C03636=1105.618,162.632,-64.067,-179.309,8.943,149.548
C03637=1105.623,162.383,-64.044,-179.311,8.940,149.548
C03638=1105.627,162.134,-64.021,-179.313,8.937,149.548
C03639=1105.632,161.885,-63.998,-179.315,8.934,149.548
C03640=1105.637,161.636,-63.975,-179.317,8.931,149.548
C03641=1105.641,161.388,-63.952,-179.319,8.928,149.547
C03642=1105.646,161.138,-63.929,-179.321,8.924,149.547
C03643=1105.650,160.890,-63.906,-179.324,8.921,149.547
C03644=1105.654,160.641,-63.883,-179.325,8.919,149.547
C03645=1105.659,160.428,-63.863,-179.327,8.916,149.547
C03646=1105.663,160.214,-63.844,-179.329,8.913,149.547
C03647=1105.667,160.001,-63.824,-179.331,8.910,149.547
C03648=1105.671,159.788,-63.804,-179.333,8.908,149.546
C03649=1105.674,159.575,-63.786,-179.335,8.905,149.546
C03650=1105.678,159.362,-63.766,-179.336,8.903,149.546
C03651=1105.682,159.148,-63.746,-179.338,8.900,149.546
C03652=1105.686,158.935,-63.727,-179.339,8.898,149.546
C03653=1105.690,158.687,-63.704,-179.342,8.894,149.546
C03654=1105.695,158.438,-63.680,-179.344,8.891,149.545
C03655=1105.700,158.189,-63.657,-179.346,8.888,149.545
C03656=1105.704,157.940,-63.635,-179.348,8.885,149.545
C03657=1105.709,157.691,-63.612,-179.350,8.881,149.545
C03658=1105.713,157.442,-63.589,-179.352,8.878,149.545
C03659=1105.718,157.193,-63.567,-179.354,8.876,149.545
C03660=1105.723,156.945,-63.544,-179.356,8.872,149.544
C03661=1105.727,156.696,-63.521,-179.358,8.869,149.544
C03662=1105.732,156.446,-63.499,-179.360,8.865,149.544
C03663=1105.736,156.197,-63.475,-179.362,8.863,149.544
C03664=1105.741,155.949,-63.454,-179.364,8.859,149.544
C03665=1105.746,155.699,-63.430,-179.366,8.856,149.543
C03666=1105.750,155.451,-63.408,-179.367,8.853,149.543
C03667=1105.756,155.202,-63.385,-179.369,8.850,149.543
C03668=1105.759,154.953,-63.363,-179.372,8.847,149.543
C03669=1105.764,154.704,-63.341,-179.374,8.843,149.543
C03670=1105.768,154.455,-63.317,-179.376,8.840,149.542
C03671=1105.773,154.206,-63.296,-179.378,8.837,149.542
C03672=1105.778,153.957,-63.272,-179.380,8.833,149.542
C03673=1105.782,153.708,-63.250,-179.382,8.830,149.542
C03674=1105.788,153.459,-63.227,-179.383,8.827,149.541
C03675=1105.792,153.210,-63.205,-179.385,8.824,149.541
C03676=1105.796,152.961,-63.182,-179.387,8.820,149.541
C03677=1105.801,152.712,-63.160,-179.389,8.817,149.541
C03678=1105.805,152.464,-63.137,-179.391,8.814,149.540
C03679=1105.810,152.214,-63.115,-179.393,8.810,149.540
